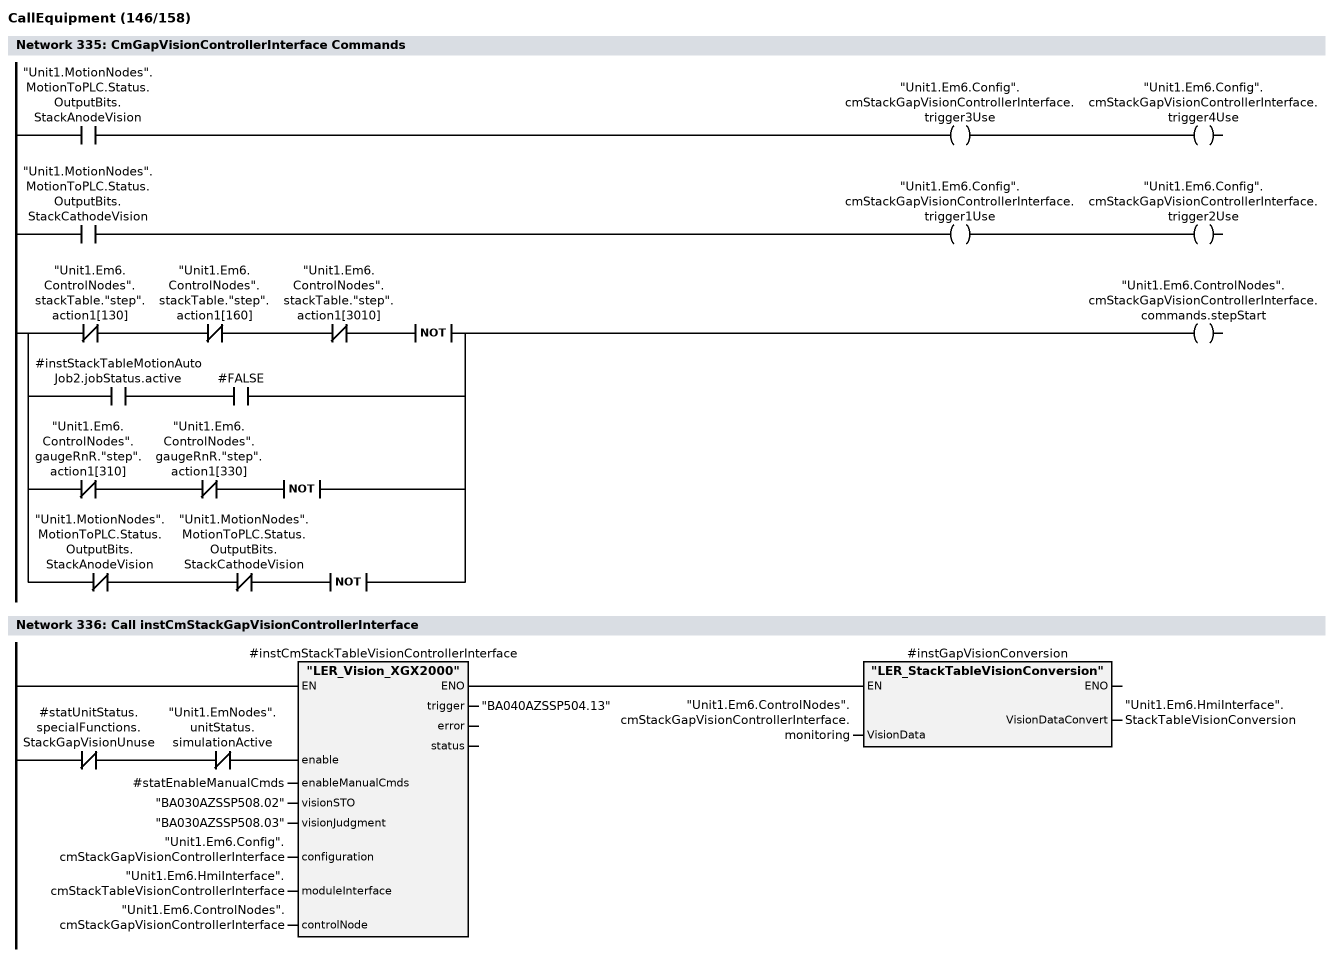
   RUNG wire#powerrail
      Contact( "Unit1.MotionNodes".MotionToPLC.Status.OutputBits.StackAnodeVision )
      Coil( "Unit1.Em6.Config".cmStackGapVisionControllerInterface.trigger3Use )
      Coil( "Unit1.Em6.Config".cmStackGapVisionControllerInterface.trigger4Use )
   END_RUNG
   RUNG wire#powerrail
      Contact( "Unit1.MotionNodes".MotionToPLC.Status.OutputBits.StackCathodeVision )
      Coil( "Unit1.Em6.Config".cmStackGapVisionControllerInterface.trigger1Use )
      Coil( "Unit1.Em6.Config".cmStackGapVisionControllerInterface.trigger2Use )
   END_RUNG
   RUNG wire#powerrail
      I_Contact( "Unit1.Em6.ControlNodes".stackTable."step".action1[130] )
      I_Contact( "Unit1.Em6.ControlNodes".stackTable."step".action1[160] )
      I_Contact( "Unit1.Em6.ControlNodes".stackTable."step".action1[3010] )
      Not()
      wire#w1
      Coil( "Unit1.Em6.ControlNodes".cmStackGapVisionControllerInterface.commands.stepStart )
   END_RUNG
   RUNG wire#powerrail
      Contact( #instStackTableMotionAutoJob2.jobStatus.active )
      Contact( #FALSE )
   END_RUNG wire#w1
   RUNG wire#powerrail
      I_Contact( "Unit1.Em6.ControlNodes".gaugeRnR."step".action1[310] )
      I_Contact( "Unit1.Em6.ControlNodes".gaugeRnR."step".action1[330] )
      Not()
   END_RUNG wire#w1
   RUNG wire#powerrail
      I_Contact( "Unit1.MotionNodes".MotionToPLC.Status.OutputBits.StackAnodeVision )
      I_Contact( "Unit1.MotionNodes".MotionToPLC.Status.OutputBits.StackCathodeVision )
      Not()
   END_RUNG wire#w1
   // the same network as SCL:
   "Unit1.Em6.Config".cmStackGapVisionControllerInterface.trigger3Use := "Unit1.MotionNodes".MotionToPLC.Status.OutputBits.StackAnodeVision;
   "Unit1.Em6.Config".cmStackGapVisionControllerInterface.trigger4Use := "Unit1.MotionNodes".MotionToPLC.Status.OutputBits.StackAnodeVision;
   "Unit1.Em6.Config".cmStackGapVisionControllerInterface.trigger1Use := "Unit1.MotionNodes".MotionToPLC.Status.OutputBits.StackCathodeVision;
   "Unit1.Em6.Config".cmStackGapVisionControllerInterface.trigger2Use := "Unit1.MotionNodes".MotionToPLC.Status.OutputBits.StackCathodeVision;
   "Unit1.Em6.ControlNodes".cmStackGapVisionControllerInterface.commands.stepStart := NOT (NOT "Unit1.Em6.ControlNodes".stackTable."step".action1[130] AND NOT "Unit1.Em6.ControlNodes".stackTable."step".action1[160] AND NOT "Unit1.Em6.ControlNodes".stackTable."step".action1[3010]) OR (#instStackTableMotionAutoJob2.jobStatus.active AND #FALSE) OR NOT (NOT "Unit1.Em6.ControlNodes".gaugeRnR."step".action1[310] AND NOT "Unit1.Em6.ControlNodes".gaugeRnR."step".action1[330]) OR NOT (NOT "Unit1.MotionNodes".MotionToPLC.Status.OutputBits.StackAnodeVision AND NOT "Unit1.MotionNodes".MotionToPLC.Status.OutputBits.StackCathodeVision);
END_REGION

REGION Network 336: Call instCmStackGapVisionControllerInterface
   RUNG wire#powerrail
      #instCmStackTableVisionControllerInterface(enable := wire#w1, enableManualCmds := #statEnableManualCmds, visionSTO := "BA030AZSSP508.02", visionJudgment := "BA030AZSSP508.03", configuration := "Unit1.Em6.Config".cmStackGapVisionControllerInterface, moduleInterface := "Unit1.Em6.HmiInterface".cmStackTableVisionControllerInterface, controlNode := "Unit1.Em6.ControlNodes".cmStackGapVisionControllerInterface, trigger => "BA040AZSSP504.13", error =>, status =>)
      #instGapVisionConversion(VisionData := "Unit1.Em6.ControlNodes".cmStackGapVisionControllerInterface.monitoring, VisionDataConvert => "Unit1.Em6.HmiInterface".StackTableVisionConversion)
   END_RUNG
   RUNG wire#powerrail
      I_Contact( #statUnitStatus.specialFunctions.StackGapVisionUnuse )
      I_Contact( "Unit1.EmNodes".unitStatus.simulationActive )
   END_RUNG wire#w1
   // the same network as SCL:
   #instCmStackTableVisionControllerInterface(enable := NOT #statUnitStatus.specialFunctions.StackGapVisionUnuse AND NOT "Unit1.EmNodes".unitStatus.simulationActive,   // "LER_Vision_XGX2000"
                           enableManualCmds := #statEnableManualCmds,
                           visionSTO := "BA030AZSSP508.02",
                           visionJudgment := "BA030AZSSP508.03",
                           configuration := "Unit1.Em6.Config".cmStackGapVisionControllerInterface,
                           moduleInterface := "Unit1.Em6.HmiInterface".cmStackTableVisionControllerInterface,
                           controlNode := "Unit1.Em6.ControlNodes".cmStackGapVisionControllerInterface,
                           trigger => "BA040AZSSP504.13",
                           ENO => #_w1);
   IF #_w1 THEN
       #instGapVisionConversion(VisionData := "Unit1.Em6.ControlNodes".cmStackGapVisionControllerInterface.monitoring,   // "LER_StackTableVisionConversion"
                               VisionDataConvert => "Unit1.Em6.HmiInterface".StackTableVisionConversion);
   END_IF;
END_REGION

REGION Network 337: *************** Feedback to Unit ***************************
END_REGION

REGION Network 338: Determine StateComplete (SC) in Mode Production
   // Conditions for the Equipment Modules "stateComplete" feedback to the unit. This feedback is given when the task in for the respective state is complete.
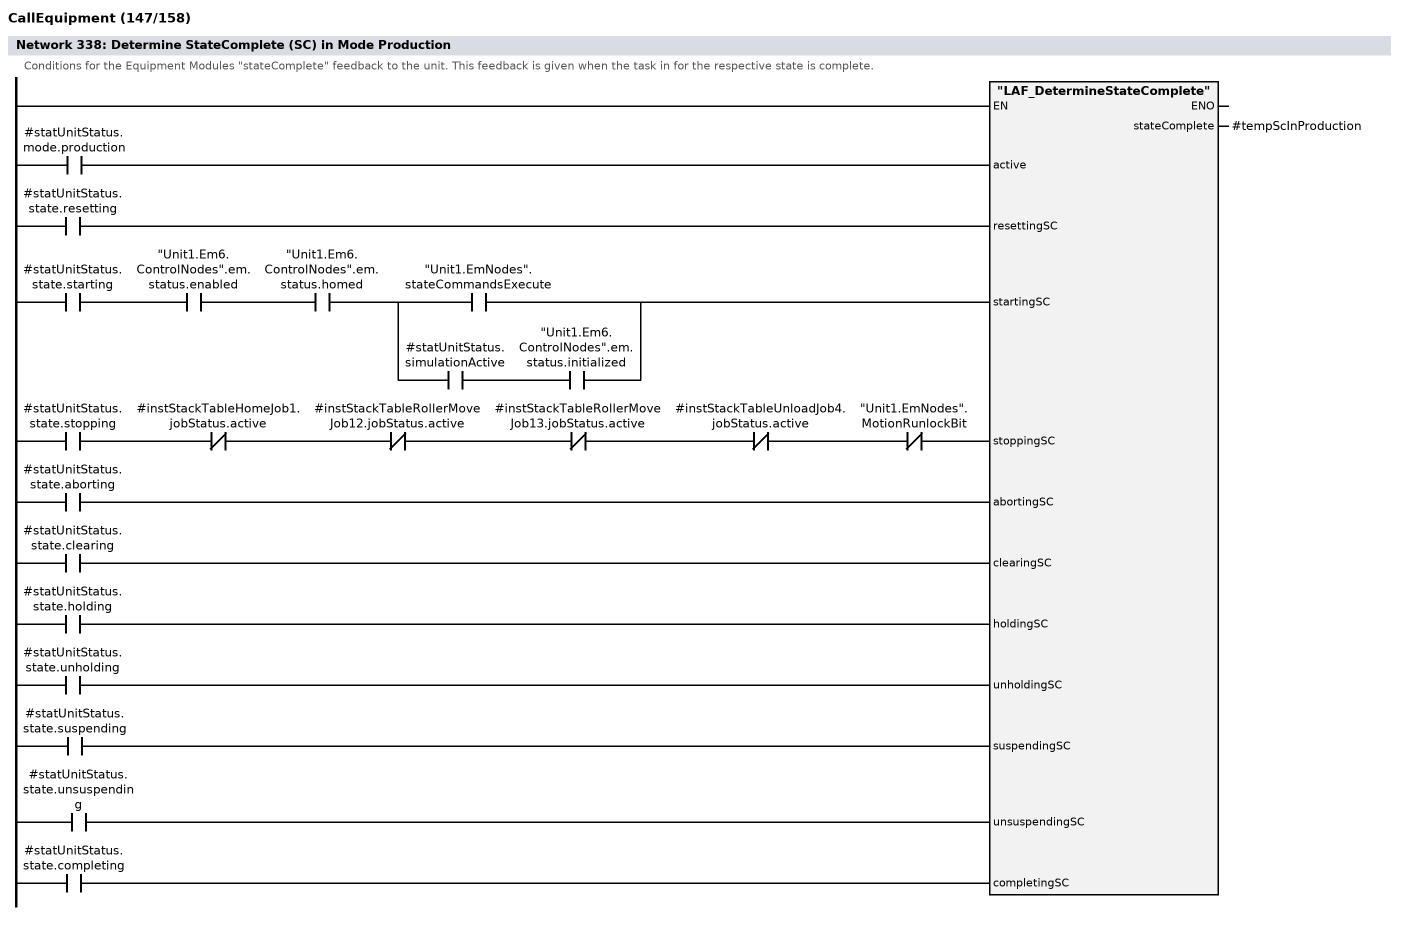
   RUNG wire#powerrail
      "LAF_DetermineStateComplete"(active := wire#w1, resettingSC := wire#w2, startingSC := wire#w4, stoppingSC := wire#w5, abortingSC := wire#w6, clearingSC := wire#w7, holdingSC := wire#w8, unholdingSC := wire#w9, suspendingSC := wire#w10, unsuspendingSC := wire#w11, completingSC := wire#w12, stateComplete => #tempScInProduction)
   END_RUNG
   RUNG wire#powerrail
      Contact( #statUnitStatus.mode.production )
   END_RUNG wire#w1
   RUNG wire#powerrail
      Contact( #statUnitStatus.state.resetting )
   END_RUNG wire#w2
   RUNG wire#powerrail
      Contact( #statUnitStatus.state.starting )
      Contact( "Unit1.Em6.ControlNodes".em.status.enabled )
      Contact( "Unit1.Em6.ControlNodes".em.status.homed )
      wire#w3
      Contact( "Unit1.EmNodes".stateCommandsExecute )
   END_RUNG wire#w4
   RUNG wire#w3
      Contact( #statUnitStatus.simulationActive )
      Contact( "Unit1.Em6.ControlNodes".em.status.initialized )
   END_RUNG wire#w4
   RUNG wire#powerrail
      Contact( #statUnitStatus.state.stopping )
      I_Contact( #instStackTableHomeJob1.jobStatus.active )
      I_Contact( #instStackTableRollerMoveJob12.jobStatus.active )
      I_Contact( #instStackTableRollerMoveJob13.jobStatus.active )
      I_Contact( #instStackTableUnloadJob4.jobStatus.active )
      I_Contact( "Unit1.EmNodes".MotionRunlockBit )
   END_RUNG wire#w5
   RUNG wire#powerrail
      Contact( #statUnitStatus.state.aborting )
   END_RUNG wire#w6
   RUNG wire#powerrail
      Contact( #statUnitStatus.state.clearing )
   END_RUNG wire#w7
   RUNG wire#powerrail
      Contact( #statUnitStatus.state.holding )
   END_RUNG wire#w8
   RUNG wire#powerrail
      Contact( #statUnitStatus.state.unholding )
   END_RUNG wire#w9
   RUNG wire#powerrail
      Contact( #statUnitStatus.state.suspending )
   END_RUNG wire#w10
   RUNG wire#powerrail
      Contact( #statUnitStatus.state.unsuspending )
   END_RUNG wire#w11
   RUNG wire#powerrail
      Contact( #statUnitStatus.state.completing )
   END_RUNG wire#w12
   // the same network as SCL:
   "LAF_DetermineStateComplete"(active := #statUnitStatus.mode.production,
                           resettingSC := #statUnitStatus.state.resetting,
                           startingSC := #statUnitStatus.state.starting AND "Unit1.Em6.ControlNodes".em.status.enabled AND "Unit1.Em6.ControlNodes".em.status.homed AND ("Unit1.EmNodes".stateCommandsExecute OR (#statUnitStatus.simulationActive AND "Unit1.Em6.ControlNodes".em.status.initialized)),
                           stoppingSC := #statUnitStatus.state.stopping AND NOT #instStackTableHomeJob1.jobStatus.active AND NOT #instStackTableRollerMoveJob12.jobStatus.active AND NOT #instStackTableRollerMoveJob13.jobStatus.active AND NOT #instStackTableUnloadJob4.jobStatus.active AND NOT "Unit1.EmNodes".MotionRunlockBit,
                           abortingSC := #statUnitStatus.state.aborting,
                           clearingSC := #statUnitStatus.state.clearing,
                           holdingSC := #statUnitStatus.state.holding,
                           unholdingSC := #statUnitStatus.state.unholding,
                           suspendingSC := #statUnitStatus.state.suspending,
                           unsuspendingSC := #statUnitStatus.state.unsuspending,
                           completingSC := #statUnitStatus.state.completing,
                           stateComplete => #tempScInProduction);
END_REGION

REGION Network 339: Determine StateComplete (SC) in Mode Maintenance/Manual
   // Conditions for the Equipment Modules "stateComplete" feedback to the unit. This feedback is given when the task in for the respective state is complete.
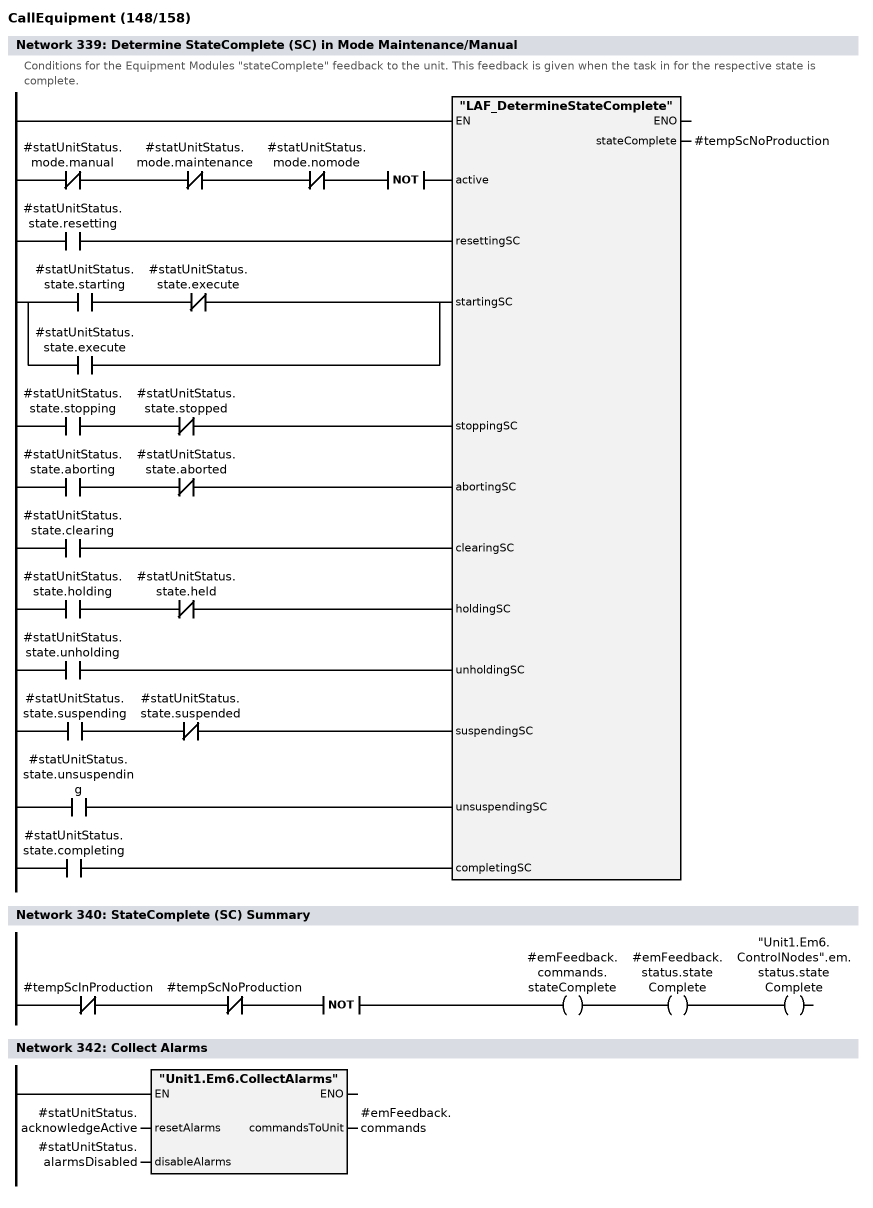
   RUNG wire#powerrail
      "LAF_DetermineStateComplete"(active := wire#w1, resettingSC := wire#w2, startingSC := wire#w3, stoppingSC := wire#w4, abortingSC := wire#w5, clearingSC := wire#w6, holdingSC := wire#w7, unholdingSC := wire#w8, suspendingSC := wire#w9, unsuspendingSC := wire#w10, completingSC := wire#w11, stateComplete => #tempScNoProduction)
   END_RUNG
   RUNG wire#powerrail
      I_Contact( #statUnitStatus.mode.manual )
      I_Contact( #statUnitStatus.mode.maintenance )
      I_Contact( #statUnitStatus.mode.nomode )
      Not()
   END_RUNG wire#w1
   RUNG wire#powerrail
      Contact( #statUnitStatus.state.resetting )
   END_RUNG wire#w2
   RUNG wire#powerrail
      Contact( #statUnitStatus.state.starting )
      I_Contact( #statUnitStatus.state.execute )
   END_RUNG wire#w3
   RUNG wire#powerrail
      Contact( #statUnitStatus.state.execute )
   END_RUNG wire#w3
   RUNG wire#powerrail
      Contact( #statUnitStatus.state.stopping )
      I_Contact( #statUnitStatus.state.stopped )
   END_RUNG wire#w4
   RUNG wire#powerrail
      Contact( #statUnitStatus.state.aborting )
      I_Contact( #statUnitStatus.state.aborted )
   END_RUNG wire#w5
   RUNG wire#powerrail
      Contact( #statUnitStatus.state.clearing )
   END_RUNG wire#w6
   RUNG wire#powerrail
      Contact( #statUnitStatus.state.holding )
      I_Contact( #statUnitStatus.state.held )
   END_RUNG wire#w7
   RUNG wire#powerrail
      Contact( #statUnitStatus.state.unholding )
   END_RUNG wire#w8
   RUNG wire#powerrail
      Contact( #statUnitStatus.state.suspending )
      I_Contact( #statUnitStatus.state.suspended )
   END_RUNG wire#w9
   RUNG wire#powerrail
      Contact( #statUnitStatus.state.unsuspending )
   END_RUNG wire#w10
   RUNG wire#powerrail
      Contact( #statUnitStatus.state.completing )
   END_RUNG wire#w11
   // the same network as SCL:
   "LAF_DetermineStateComplete"(active := NOT (NOT #statUnitStatus.mode.manual AND NOT #statUnitStatus.mode.maintenance AND NOT #statUnitStatus.mode.nomode),
                           resettingSC := #statUnitStatus.state.resetting,
                           startingSC := (#statUnitStatus.state.starting AND NOT #statUnitStatus.state.execute) OR #statUnitStatus.state.execute,
                           stoppingSC := #statUnitStatus.state.stopping AND NOT #statUnitStatus.state.stopped,
                           abortingSC := #statUnitStatus.state.aborting AND NOT #statUnitStatus.state.aborted,
                           clearingSC := #statUnitStatus.state.clearing,
                           holdingSC := #statUnitStatus.state.holding AND NOT #statUnitStatus.state.held,
                           unholdingSC := #statUnitStatus.state.unholding,
                           suspendingSC := #statUnitStatus.state.suspending AND NOT #statUnitStatus.state.suspended,
                           unsuspendingSC := #statUnitStatus.state.unsuspending,
                           completingSC := #statUnitStatus.state.completing,
                           stateComplete => #tempScNoProduction);
END_REGION

REGION Network 340: StateComplete (SC) Summary
   RUNG wire#powerrail
      I_Contact( #tempScInProduction )
      I_Contact( #tempScNoProduction )
      Not()
      Coil( #emFeedback.commands.stateComplete )
      Coil( #emFeedback.status.stateComplete )
      Coil( "Unit1.Em6.ControlNodes".em.status.stateComplete )
   END_RUNG
   // the same network as SCL:
   #emFeedback.commands.stateComplete := NOT (NOT #tempScInProduction AND NOT #tempScNoProduction);
   #emFeedback.status.stateComplete := #emFeedback.commands.stateComplete;
   "Unit1.Em6.ControlNodes".em.status.stateComplete := #emFeedback.commands.stateComplete;
END_REGION

REGION Network 341: *************** Alarms **********************************
END_REGION

REGION Network 342: Collect Alarms
   RUNG wire#powerrail
      "Unit1.Em6.CollectAlarms"(resetAlarms := #statUnitStatus.acknowledgeActive, disableAlarms := #statUnitStatus.alarmsDisabled, commandsToUnit => #emFeedback.commands)
   END_RUNG
   // the same network as SCL:
   "Unit1.Em6.CollectAlarms"(resetAlarms := #statUnitStatus.acknowledgeActive,
                           disableAlarms := #statUnitStatus.alarmsDisabled,
                           commandsToUnit => #emFeedback.commands);
END_REGION

REGION Network 343: Manage Alarms
   // Derive commands from the ProDiag supervision. The ProDiag supervisions contain categories which define the reaction of these supervisions (e.g. abort, stop, hold). These are handed over as commands to the unit level.
   // Alternatively, if no ProDiag should be used, you can use the LAF_ManageBitAlarms to realize bit alarm handling. This block can be found in LAF in folder 70_AlarmHandling.
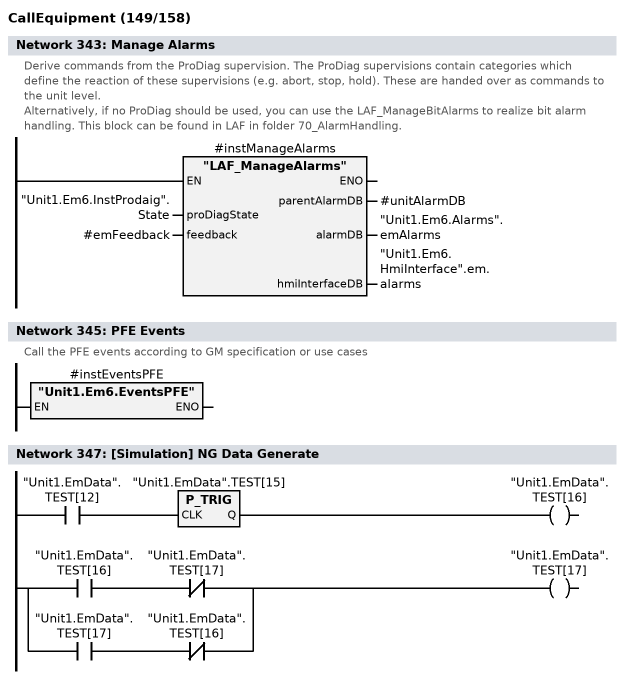
   RUNG wire#powerrail
      #instManageAlarms(proDiagState := "Unit1.Em6.InstProdaig".State, feedback := #emFeedback, parentAlarmDB => #unitAlarmDB, alarmDB => "Unit1.Em6.Alarms".emAlarms, hmiInterfaceDB => "Unit1.Em6.HmiInterface".em.alarms)
   END_RUNG
   // the same network as SCL:
   #instManageAlarms(proDiagState := "Unit1.Em6.InstProdaig".State,   // "LAF_ManageAlarms"
                     feedback := #emFeedback,
                     parentAlarmDB => #unitAlarmDB,
                     alarmDB => "Unit1.Em6.Alarms".emAlarms,
                     hmiInterfaceDB => "Unit1.Em6.HmiInterface".em.alarms);
END_REGION

REGION Network 344: *************** PFE Events**********************************
END_REGION

REGION Network 345: PFE Events
   // Call the PFE events according to GM specification or use cases
   RUNG wire#powerrail
      #instEventsPFE()
   END_RUNG
   // the same network as SCL:
   #instEventsPFE();   // "Unit1.Em6.EventsPFE"
END_REGION

REGION Network 346: ******************** Part Data ********************
END_REGION

REGION Network 347: [Simulation] NG Data Generate
   RUNG wire#powerrail
      Contact( "Unit1.EmData".TEST[12] )
      P_Trig( "Unit1.EmData".TEST[15] )
      Coil( "Unit1.EmData".TEST[16] )
   END_RUNG
   RUNG wire#powerrail
      Contact( "Unit1.EmData".TEST[16] )
      I_Contact( "Unit1.EmData".TEST[17] )
      wire#w1
      Coil( "Unit1.EmData".TEST[17] )
   END_RUNG
   RUNG wire#powerrail
      Contact( "Unit1.EmData".TEST[17] )
      I_Contact( "Unit1.EmData".TEST[16] )
   END_RUNG wire#w1
   // the same network as SCL:
   #_w1 := "Unit1.EmData".TEST[12];
   #_w2 := #_w1 AND NOT "Unit1.EmData".TEST[15];   // rising edge
   "Unit1.EmData".TEST[15] := #_w1;
   "Unit1.EmData".TEST[16] := #_w2;
   "Unit1.EmData".TEST[17] := ("Unit1.EmData".TEST[16] AND NOT "Unit1.EmData".TEST[17]) OR ("Unit1.EmData".TEST[17] AND NOT "Unit1.EmData".TEST[16]);
END_REGION

REGION Network 348: Gap Vision Data
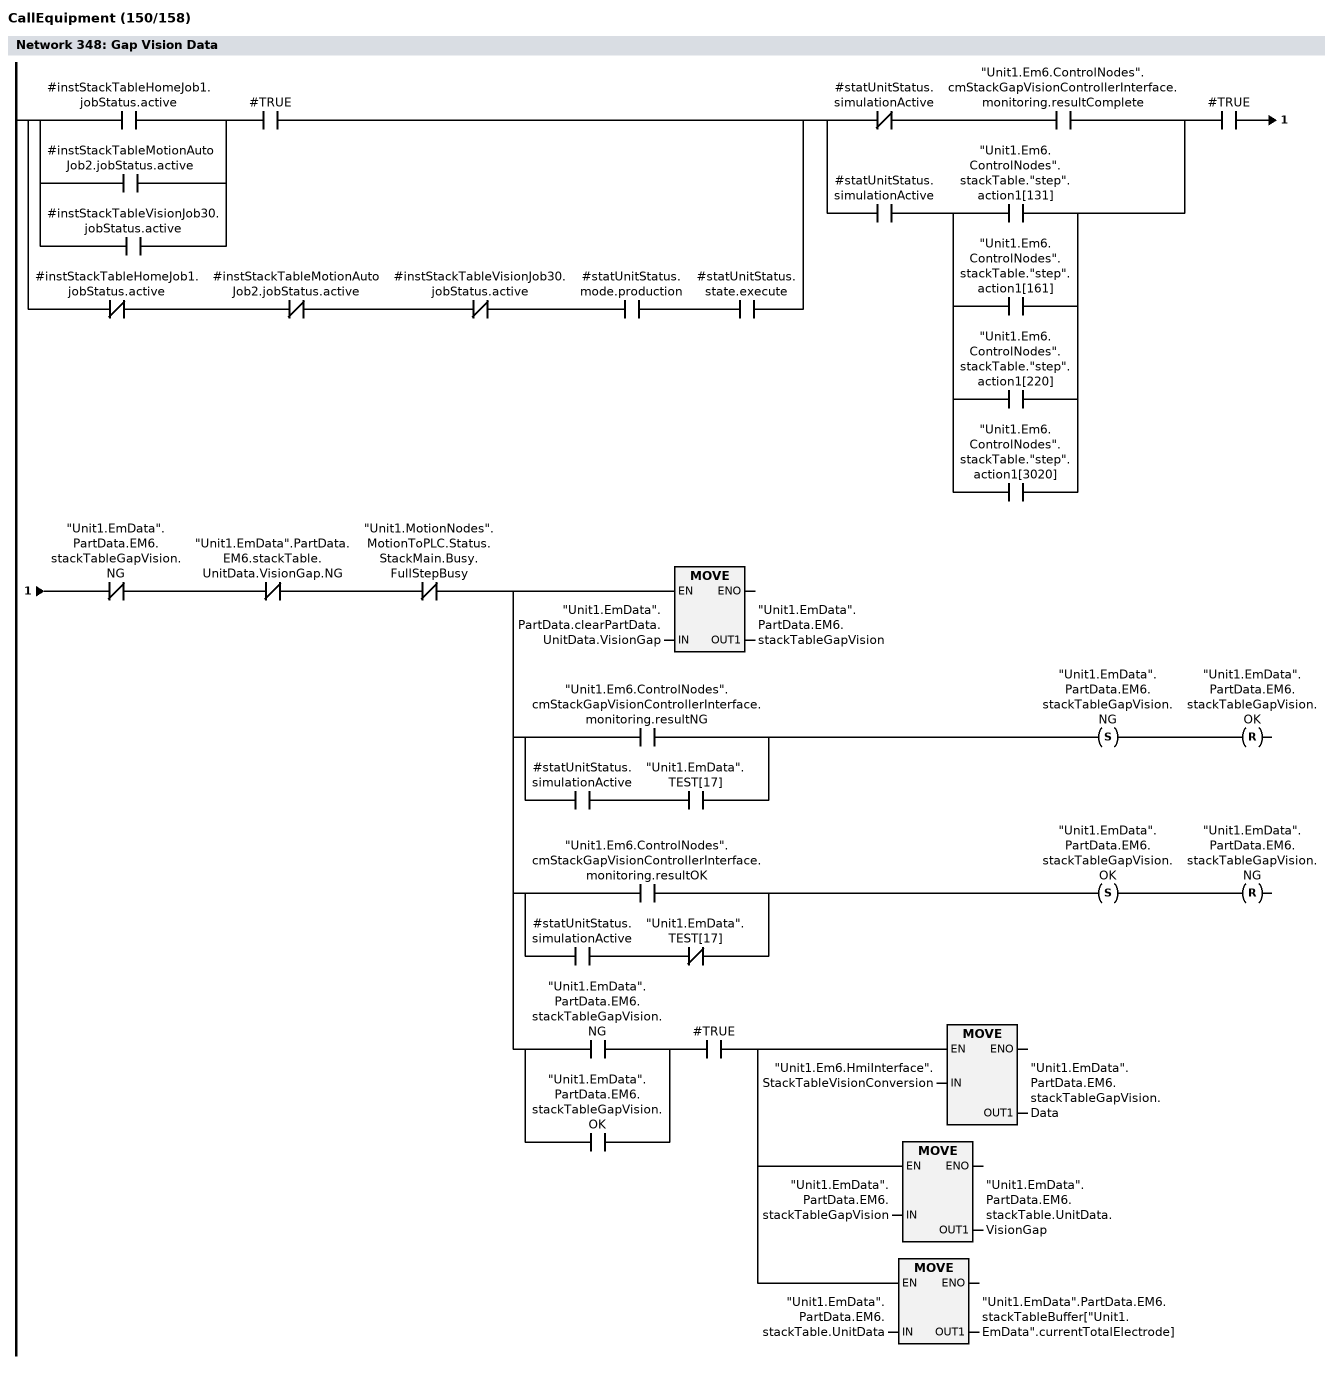
   RUNG wire#powerrail
      Contact( #instStackTableHomeJob1.jobStatus.active )
      wire#w1
      Contact( #TRUE )
      wire#w2
      I_Contact( #statUnitStatus.simulationActive )
      Contact( "Unit1.Em6.ControlNodes".cmStackGapVisionControllerInterface.monitoring.resultComplete )
      wire#w3
      Contact( #TRUE )
      I_Contact( "Unit1.EmData".PartData.EM6.stackTableGapVision.NG )
      I_Contact( "Unit1.EmData".PartData.EM6.stackTable.UnitData.VisionGap.NG )
      I_Contact( "Unit1.MotionNodes".MotionToPLC.Status.StackMain.Busy.FullStepBusy )
      wire#w5
      Move(in := "Unit1.EmData".PartData.clearPartData.UnitData.VisionGap, out1 => "Unit1.EmData".PartData.EM6.stackTableGapVision)
   END_RUNG
   RUNG wire#powerrail
      Contact( #instStackTableMotionAutoJob2.jobStatus.active )
   END_RUNG wire#w1
   RUNG wire#powerrail
      Contact( #instStackTableVisionJob30.jobStatus.active )
   END_RUNG wire#w1
   RUNG wire#powerrail
      I_Contact( #instStackTableHomeJob1.jobStatus.active )
      I_Contact( #instStackTableMotionAutoJob2.jobStatus.active )
      I_Contact( #instStackTableVisionJob30.jobStatus.active )
      Contact( #statUnitStatus.mode.production )
      Contact( #statUnitStatus.state.execute )
   END_RUNG wire#w2
   RUNG wire#w2
      Contact( #statUnitStatus.simulationActive )
      wire#w4
      Contact( "Unit1.Em6.ControlNodes".stackTable."step".action1[131] )
   END_RUNG wire#w3
   RUNG wire#w4
      Contact( "Unit1.Em6.ControlNodes".stackTable."step".action1[161] )
   END_RUNG wire#w3
   RUNG wire#w4
      Contact( "Unit1.Em6.ControlNodes".stackTable."step".action1[220] )
   END_RUNG wire#w3
   RUNG wire#w4
      Contact( "Unit1.Em6.ControlNodes".stackTable."step".action1[3020] )
   END_RUNG wire#w3
   RUNG wire#w5
      Contact( "Unit1.Em6.ControlNodes".cmStackGapVisionControllerInterface.monitoring.resultNG )
      wire#w6
      S_Coil( "Unit1.EmData".PartData.EM6.stackTableGapVision.NG )
      R_Coil( "Unit1.EmData".PartData.EM6.stackTableGapVision.OK )
   END_RUNG
   RUNG wire#w5
      Contact( #statUnitStatus.simulationActive )
      Contact( "Unit1.EmData".TEST[17] )
   END_RUNG wire#w6
   RUNG wire#w5
      Contact( "Unit1.Em6.ControlNodes".cmStackGapVisionControllerInterface.monitoring.resultOK )
      wire#w7
      S_Coil( "Unit1.EmData".PartData.EM6.stackTableGapVision.OK )
      R_Coil( "Unit1.EmData".PartData.EM6.stackTableGapVision.NG )
   END_RUNG
   RUNG wire#w5
      Contact( #statUnitStatus.simulationActive )
      I_Contact( "Unit1.EmData".TEST[17] )
   END_RUNG wire#w7
   RUNG wire#w5
      Contact( "Unit1.EmData".PartData.EM6.stackTableGapVision.NG )
      wire#w8
      Contact( #TRUE )
      wire#w9
      Move(in := "Unit1.Em6.HmiInterface".StackTableVisionConversion, out1 => "Unit1.EmData".PartData.EM6.stackTableGapVision.Data)
   END_RUNG
   RUNG wire#w5
      Contact( "Unit1.EmData".PartData.EM6.stackTableGapVision.OK )
   END_RUNG wire#w8
   RUNG wire#w9
      Move(in := "Unit1.EmData".PartData.EM6.stackTableGapVision, out1 => "Unit1.EmData".PartData.EM6.stackTable.UnitData.VisionGap)
   END_RUNG
   RUNG wire#w9
      Move(in := "Unit1.EmData".PartData.EM6.stackTable.UnitData, out1 => "Unit1.EmData".PartData.EM6.stackTableBuffer["Unit1.EmData".currentTotalElectrode])
   END_RUNG
   // the same network as SCL:
   #_w1 := (((#instStackTableHomeJob1.jobStatus.active OR #instStackTableMotionAutoJob2.jobStatus.active OR #instStackTableVisionJob30.jobStatus.active) AND #TRUE) OR (NOT #instStackTableHomeJob1.jobStatus.active AND NOT #instStackTableMotionAutoJob2.jobStatus.active AND NOT #instStackTableVisionJob30.jobStatus.active AND #statUnitStatus.mode.production AND #statUnitStatus.state.execute)) AND ((NOT #statUnitStatus.simulationActive AND "Unit1.Em6.ControlNodes".cmStackGapVisionControllerInterface.monitoring.resultComplete) OR (#statUnitStatus.simulationActive AND ("Unit1.Em6.ControlNodes".stackTable."step".action1[131] OR "Unit1.Em6.ControlNodes".stackTable."step".action1[161] OR "Unit1.Em6.ControlNodes".stackTable."step".action1[220] OR "Unit1.Em6.ControlNodes".stackTable."step".action1[3020]))) AND #TRUE AND NOT "Unit1.EmData".PartData.EM6.stackTableGapVision.NG AND NOT "Unit1.EmData".PartData.EM6.stackTable.UnitData.VisionGap.NG AND NOT "Unit1.MotionNodes".MotionToPLC.Status.StackMain.Busy.FullStepBusy;
   IF #_w1 THEN
       "Unit1.EmData".PartData.EM6.stackTableGapVision := "Unit1.EmData".PartData.clearPartData.UnitData.VisionGap;
   END_IF;
   IF #_w1 AND ("Unit1.Em6.ControlNodes".cmStackGapVisionControllerInterface.monitoring.resultNG OR (#statUnitStatus.simulationActive AND "Unit1.EmData".TEST[17])) THEN
       "Unit1.EmData".PartData.EM6.stackTableGapVision.NG := TRUE;
       "Unit1.EmData".PartData.EM6.stackTableGapVision.OK := FALSE;
   END_IF;
   IF #_w1 AND ("Unit1.Em6.ControlNodes".cmStackGapVisionControllerInterface.monitoring.resultOK OR (#statUnitStatus.simulationActive AND NOT "Unit1.EmData".TEST[17])) THEN
       "Unit1.EmData".PartData.EM6.stackTableGapVision.OK := TRUE;
       "Unit1.EmData".PartData.EM6.stackTableGapVision.NG := FALSE;
   END_IF;
   IF #_w1 AND ("Unit1.EmData".PartData.EM6.stackTableGapVision.NG OR "Unit1.EmData".PartData.EM6.stackTableGapVision.OK) AND #TRUE THEN
       "Unit1.EmData".PartData.EM6.stackTableGapVision.Data := "Unit1.Em6.HmiInterface".StackTableVisionConversion;
       "Unit1.EmData".PartData.EM6.stackTable.UnitData.VisionGap := "Unit1.EmData".PartData.EM6.stackTableGapVision;
       "Unit1.EmData".PartData.EM6.stackTableBuffer["Unit1.EmData".currentTotalElectrode] := "Unit1.EmData".PartData.EM6.stackTable.UnitData;
   END_IF;
END_REGION

REGION Network 349: ******************** Map 64Pos Positiotion ********************
END_REGION

REGION Network 350: StackTableAxis Z Postion [1] Mapping
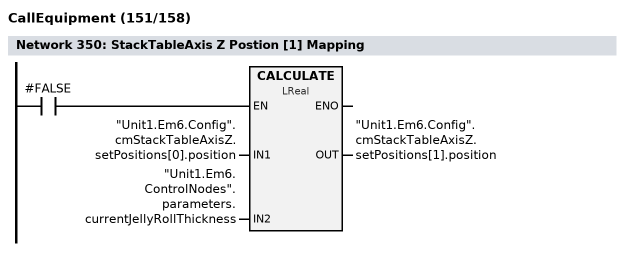
   RUNG wire#powerrail
      Contact( #FALSE )
      { S7_Templates := "SrcType := LReal"; S7_Expression := "IN1 + IN2" } Calculate(in1 := "Unit1.Em6.Config".cmStackTableAxisZ.setPositions[0].position, in2 := "Unit1.Em6.ControlNodes".parameters.currentJellyRollThickness, out => "Unit1.Em6.Config".cmStackTableAxisZ.setPositions[1].position)
   END_RUNG
   // the same network as SCL:
   IF #FALSE THEN
       "Unit1.Em6.Config".cmStackTableAxisZ.setPositions[1].position := "Unit1.Em6.Config".cmStackTableAxisZ.setPositions[0].position + "Unit1.Em6.ControlNodes".parameters.currentJellyRollThickness;
   END_IF;
END_REGION

REGION Network 351: ******************** Unit Output ********************
END_REGION

REGION Network 352: Em Nodes Brake Test
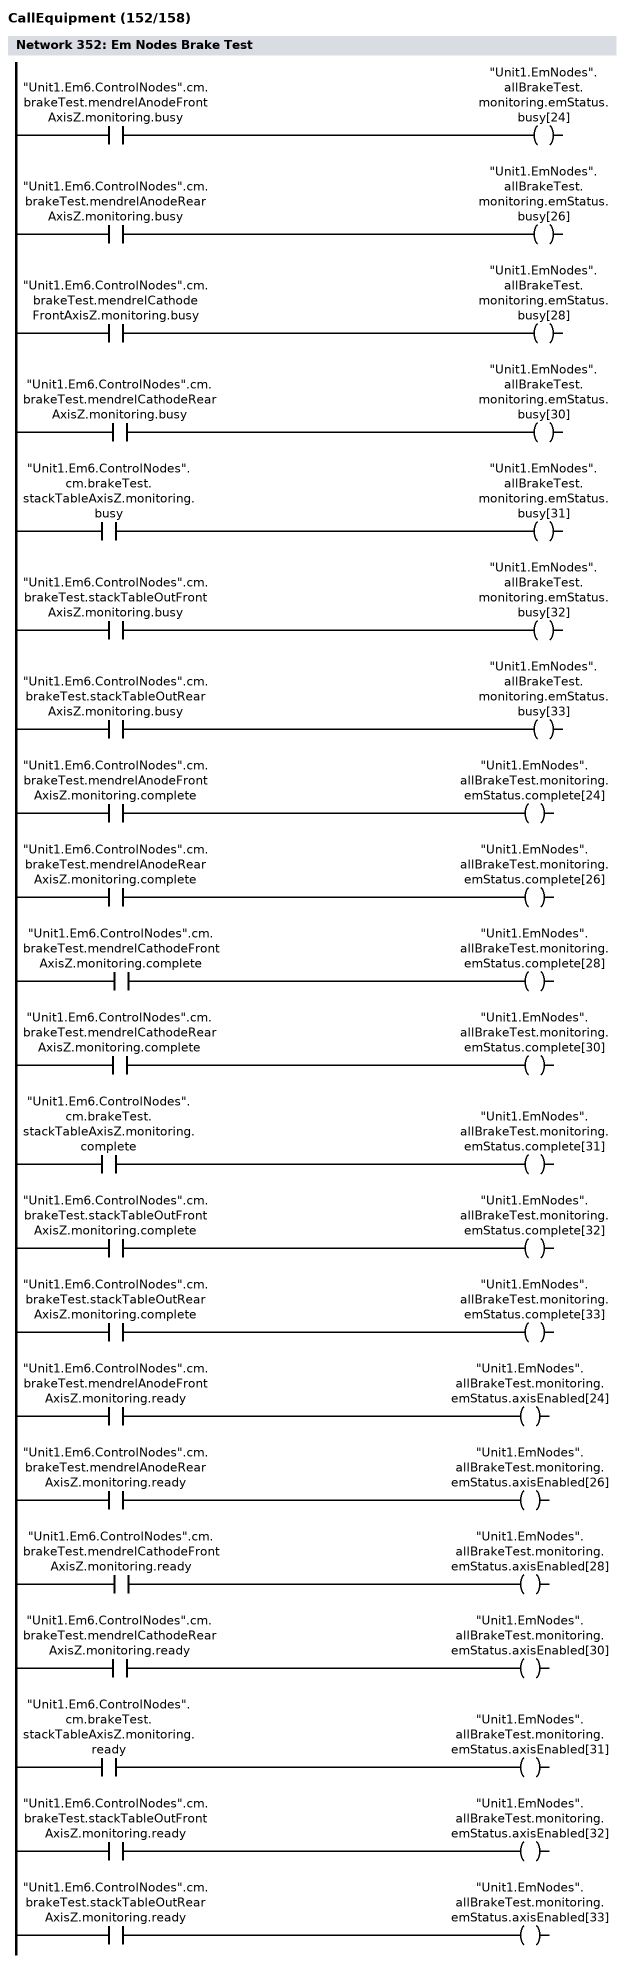
   RUNG wire#powerrail
      Contact( "Unit1.Em6.ControlNodes".cm.brakeTest.mendrelAnodeFrontAxisZ.monitoring.busy )
      Coil( "Unit1.EmNodes".allBrakeTest.monitoring.emStatus.busy[24] )
   END_RUNG
   RUNG wire#powerrail
      Contact( "Unit1.Em6.ControlNodes".cm.brakeTest.mendrelAnodeRearAxisZ.monitoring.busy )
      Coil( "Unit1.EmNodes".allBrakeTest.monitoring.emStatus.busy[26] )
   END_RUNG
   RUNG wire#powerrail
      Contact( "Unit1.Em6.ControlNodes".cm.brakeTest.mendrelCathodeFrontAxisZ.monitoring.busy )
      Coil( "Unit1.EmNodes".allBrakeTest.monitoring.emStatus.busy[28] )
   END_RUNG
   RUNG wire#powerrail
      Contact( "Unit1.Em6.ControlNodes".cm.brakeTest.mendrelCathodeRearAxisZ.monitoring.busy )
      Coil( "Unit1.EmNodes".allBrakeTest.monitoring.emStatus.busy[30] )
   END_RUNG
   RUNG wire#powerrail
      Contact( "Unit1.Em6.ControlNodes".cm.brakeTest.stackTableAxisZ.monitoring.busy )
      Coil( "Unit1.EmNodes".allBrakeTest.monitoring.emStatus.busy[31] )
   END_RUNG
   RUNG wire#powerrail
      Contact( "Unit1.Em6.ControlNodes".cm.brakeTest.stackTableOutFrontAxisZ.monitoring.busy )
      Coil( "Unit1.EmNodes".allBrakeTest.monitoring.emStatus.busy[32] )
   END_RUNG
   RUNG wire#powerrail
      Contact( "Unit1.Em6.ControlNodes".cm.brakeTest.stackTableOutRearAxisZ.monitoring.busy )
      Coil( "Unit1.EmNodes".allBrakeTest.monitoring.emStatus.busy[33] )
   END_RUNG
   RUNG wire#powerrail
      Contact( "Unit1.Em6.ControlNodes".cm.brakeTest.mendrelAnodeFrontAxisZ.monitoring.complete )
      Coil( "Unit1.EmNodes".allBrakeTest.monitoring.emStatus.complete[24] )
   END_RUNG
   RUNG wire#powerrail
      Contact( "Unit1.Em6.ControlNodes".cm.brakeTest.mendrelAnodeRearAxisZ.monitoring.complete )
      Coil( "Unit1.EmNodes".allBrakeTest.monitoring.emStatus.complete[26] )
   END_RUNG
   RUNG wire#powerrail
      Contact( "Unit1.Em6.ControlNodes".cm.brakeTest.mendrelCathodeFrontAxisZ.monitoring.complete )
      Coil( "Unit1.EmNodes".allBrakeTest.monitoring.emStatus.complete[28] )
   END_RUNG
   RUNG wire#powerrail
      Contact( "Unit1.Em6.ControlNodes".cm.brakeTest.mendrelCathodeRearAxisZ.monitoring.complete )
      Coil( "Unit1.EmNodes".allBrakeTest.monitoring.emStatus.complete[30] )
   END_RUNG
   RUNG wire#powerrail
      Contact( "Unit1.Em6.ControlNodes".cm.brakeTest.stackTableAxisZ.monitoring.complete )
      Coil( "Unit1.EmNodes".allBrakeTest.monitoring.emStatus.complete[31] )
   END_RUNG
   RUNG wire#powerrail
      Contact( "Unit1.Em6.ControlNodes".cm.brakeTest.stackTableOutFrontAxisZ.monitoring.complete )
      Coil( "Unit1.EmNodes".allBrakeTest.monitoring.emStatus.complete[32] )
   END_RUNG
   RUNG wire#powerrail
      Contact( "Unit1.Em6.ControlNodes".cm.brakeTest.stackTableOutRearAxisZ.monitoring.complete )
      Coil( "Unit1.EmNodes".allBrakeTest.monitoring.emStatus.complete[33] )
   END_RUNG
   RUNG wire#powerrail
      Contact( "Unit1.Em6.ControlNodes".cm.brakeTest.mendrelAnodeFrontAxisZ.monitoring.ready )
      Coil( "Unit1.EmNodes".allBrakeTest.monitoring.emStatus.axisEnabled[24] )
   END_RUNG
   RUNG wire#powerrail
      Contact( "Unit1.Em6.ControlNodes".cm.brakeTest.mendrelAnodeRearAxisZ.monitoring.ready )
      Coil( "Unit1.EmNodes".allBrakeTest.monitoring.emStatus.axisEnabled[26] )
   END_RUNG
   RUNG wire#powerrail
      Contact( "Unit1.Em6.ControlNodes".cm.brakeTest.mendrelCathodeFrontAxisZ.monitoring.ready )
      Coil( "Unit1.EmNodes".allBrakeTest.monitoring.emStatus.axisEnabled[28] )
   END_RUNG
   RUNG wire#powerrail
      Contact( "Unit1.Em6.ControlNodes".cm.brakeTest.mendrelCathodeRearAxisZ.monitoring.ready )
      Coil( "Unit1.EmNodes".allBrakeTest.monitoring.emStatus.axisEnabled[30] )
   END_RUNG
   RUNG wire#powerrail
      Contact( "Unit1.Em6.ControlNodes".cm.brakeTest.stackTableAxisZ.monitoring.ready )
      Coil( "Unit1.EmNodes".allBrakeTest.monitoring.emStatus.axisEnabled[31] )
   END_RUNG
   RUNG wire#powerrail
      Contact( "Unit1.Em6.ControlNodes".cm.brakeTest.stackTableOutFrontAxisZ.monitoring.ready )
      Coil( "Unit1.EmNodes".allBrakeTest.monitoring.emStatus.axisEnabled[32] )
   END_RUNG
   RUNG wire#powerrail
      Contact( "Unit1.Em6.ControlNodes".cm.brakeTest.stackTableOutRearAxisZ.monitoring.ready )
      Coil( "Unit1.EmNodes".allBrakeTest.monitoring.emStatus.axisEnabled[33] )
   END_RUNG
   // the same network as SCL:
   "Unit1.EmNodes".allBrakeTest.monitoring.emStatus.busy[24] := "Unit1.Em6.ControlNodes".cm.brakeTest.mendrelAnodeFrontAxisZ.monitoring.busy;
   "Unit1.EmNodes".allBrakeTest.monitoring.emStatus.busy[26] := "Unit1.Em6.ControlNodes".cm.brakeTest.mendrelAnodeRearAxisZ.monitoring.busy;
   "Unit1.EmNodes".allBrakeTest.monitoring.emStatus.busy[28] := "Unit1.Em6.ControlNodes".cm.brakeTest.mendrelCathodeFrontAxisZ.monitoring.busy;
   "Unit1.EmNodes".allBrakeTest.monitoring.emStatus.busy[30] := "Unit1.Em6.ControlNodes".cm.brakeTest.mendrelCathodeRearAxisZ.monitoring.busy;
   "Unit1.EmNodes".allBrakeTest.monitoring.emStatus.busy[31] := "Unit1.Em6.ControlNodes".cm.brakeTest.stackTableAxisZ.monitoring.busy;
   "Unit1.EmNodes".allBrakeTest.monitoring.emStatus.busy[32] := "Unit1.Em6.ControlNodes".cm.brakeTest.stackTableOutFrontAxisZ.monitoring.busy;
   "Unit1.EmNodes".allBrakeTest.monitoring.emStatus.busy[33] := "Unit1.Em6.ControlNodes".cm.brakeTest.stackTableOutRearAxisZ.monitoring.busy;
   "Unit1.EmNodes".allBrakeTest.monitoring.emStatus.complete[24] := "Unit1.Em6.ControlNodes".cm.brakeTest.mendrelAnodeFrontAxisZ.monitoring.complete;
   "Unit1.EmNodes".allBrakeTest.monitoring.emStatus.complete[26] := "Unit1.Em6.ControlNodes".cm.brakeTest.mendrelAnodeRearAxisZ.monitoring.complete;
   "Unit1.EmNodes".allBrakeTest.monitoring.emStatus.complete[28] := "Unit1.Em6.ControlNodes".cm.brakeTest.mendrelCathodeFrontAxisZ.monitoring.complete;
   "Unit1.EmNodes".allBrakeTest.monitoring.emStatus.complete[30] := "Unit1.Em6.ControlNodes".cm.brakeTest.mendrelCathodeRearAxisZ.monitoring.complete;
   "Unit1.EmNodes".allBrakeTest.monitoring.emStatus.complete[31] := "Unit1.Em6.ControlNodes".cm.brakeTest.stackTableAxisZ.monitoring.complete;
   "Unit1.EmNodes".allBrakeTest.monitoring.emStatus.complete[32] := "Unit1.Em6.ControlNodes".cm.brakeTest.stackTableOutFrontAxisZ.monitoring.complete;
   "Unit1.EmNodes".allBrakeTest.monitoring.emStatus.complete[33] := "Unit1.Em6.ControlNodes".cm.brakeTest.stackTableOutRearAxisZ.monitoring.complete;
   "Unit1.EmNodes".allBrakeTest.monitoring.emStatus.axisEnabled[24] := "Unit1.Em6.ControlNodes".cm.brakeTest.mendrelAnodeFrontAxisZ.monitoring.ready;
   "Unit1.EmNodes".allBrakeTest.monitoring.emStatus.axisEnabled[26] := "Unit1.Em6.ControlNodes".cm.brakeTest.mendrelAnodeRearAxisZ.monitoring.ready;
   "Unit1.EmNodes".allBrakeTest.monitoring.emStatus.axisEnabled[28] := "Unit1.Em6.ControlNodes".cm.brakeTest.mendrelCathodeFrontAxisZ.monitoring.ready;
   "Unit1.EmNodes".allBrakeTest.monitoring.emStatus.axisEnabled[30] := "Unit1.Em6.ControlNodes".cm.brakeTest.mendrelCathodeRearAxisZ.monitoring.ready;
   "Unit1.EmNodes".allBrakeTest.monitoring.emStatus.axisEnabled[31] := "Unit1.Em6.ControlNodes".cm.brakeTest.stackTableAxisZ.monitoring.ready;
   "Unit1.EmNodes".allBrakeTest.monitoring.emStatus.axisEnabled[32] := "Unit1.Em6.ControlNodes".cm.brakeTest.stackTableOutFrontAxisZ.monitoring.ready;
   "Unit1.EmNodes".allBrakeTest.monitoring.emStatus.axisEnabled[33] := "Unit1.Em6.ControlNodes".cm.brakeTest.stackTableOutRearAxisZ.monitoring.ready;
END_REGION

REGION Network 353: Em Relations Home Check
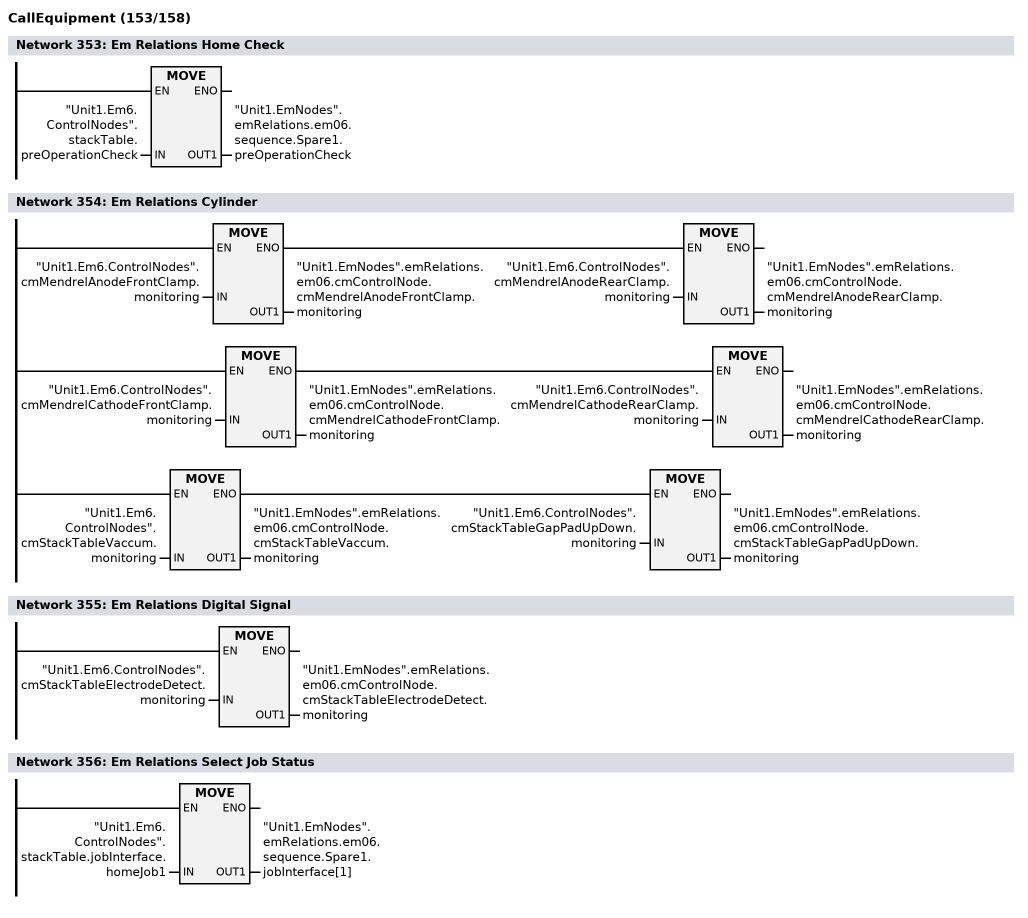
   RUNG wire#powerrail
      Move(in := "Unit1.Em6.ControlNodes".stackTable.preOperationCheck, out1 => "Unit1.EmNodes".emRelations.em06.sequence.Spare1.preOperationCheck)
   END_RUNG
   // the same network as SCL:
   "Unit1.EmNodes".emRelations.em06.sequence.Spare1.preOperationCheck := "Unit1.Em6.ControlNodes".stackTable.preOperationCheck;
END_REGION

REGION Network 354: Em Relations Cylinder
   RUNG wire#powerrail
      Move(in := "Unit1.Em6.ControlNodes".cmMendrelAnodeFrontClamp.monitoring, out1 => "Unit1.EmNodes".emRelations.em06.cmControlNode.cmMendrelAnodeFrontClamp.monitoring)
      Move(in := "Unit1.Em6.ControlNodes".cmMendrelAnodeRearClamp.monitoring, out1 => "Unit1.EmNodes".emRelations.em06.cmControlNode.cmMendrelAnodeRearClamp.monitoring)
   END_RUNG
   RUNG wire#powerrail
      Move(in := "Unit1.Em6.ControlNodes".cmMendrelCathodeFrontClamp.monitoring, out1 => "Unit1.EmNodes".emRelations.em06.cmControlNode.cmMendrelCathodeFrontClamp.monitoring)
      Move(in := "Unit1.Em6.ControlNodes".cmMendrelCathodeRearClamp.monitoring, out1 => "Unit1.EmNodes".emRelations.em06.cmControlNode.cmMendrelCathodeRearClamp.monitoring)
   END_RUNG
   RUNG wire#powerrail
      Move(in := "Unit1.Em6.ControlNodes".cmStackTableVaccum.monitoring, out1 => "Unit1.EmNodes".emRelations.em06.cmControlNode.cmStackTableVaccum.monitoring)
      Move(in := "Unit1.Em6.ControlNodes".cmStackTableGapPadUpDown.monitoring, out1 => "Unit1.EmNodes".emRelations.em06.cmControlNode.cmStackTableGapPadUpDown.monitoring)
   END_RUNG
   // the same network as SCL:
   "Unit1.EmNodes".emRelations.em06.cmControlNode.cmMendrelAnodeFrontClamp.monitoring := "Unit1.Em6.ControlNodes".cmMendrelAnodeFrontClamp.monitoring;
   "Unit1.EmNodes".emRelations.em06.cmControlNode.cmMendrelAnodeRearClamp.monitoring := "Unit1.Em6.ControlNodes".cmMendrelAnodeRearClamp.monitoring;
   "Unit1.EmNodes".emRelations.em06.cmControlNode.cmMendrelCathodeFrontClamp.monitoring := "Unit1.Em6.ControlNodes".cmMendrelCathodeFrontClamp.monitoring;
   "Unit1.EmNodes".emRelations.em06.cmControlNode.cmMendrelCathodeRearClamp.monitoring := "Unit1.Em6.ControlNodes".cmMendrelCathodeRearClamp.monitoring;
   "Unit1.EmNodes".emRelations.em06.cmControlNode.cmStackTableVaccum.monitoring := "Unit1.Em6.ControlNodes".cmStackTableVaccum.monitoring;
   "Unit1.EmNodes".emRelations.em06.cmControlNode.cmStackTableGapPadUpDown.monitoring := "Unit1.Em6.ControlNodes".cmStackTableGapPadUpDown.monitoring;
END_REGION

REGION Network 355: Em Relations Digital Signal
   RUNG wire#powerrail
      Move(in := "Unit1.Em6.ControlNodes".cmStackTableElectrodeDetect.monitoring, out1 => "Unit1.EmNodes".emRelations.em06.cmControlNode.cmStackTableElectrodeDetect.monitoring)
   END_RUNG
   // the same network as SCL:
   "Unit1.EmNodes".emRelations.em06.cmControlNode.cmStackTableElectrodeDetect.monitoring := "Unit1.Em6.ControlNodes".cmStackTableElectrodeDetect.monitoring;
END_REGION

REGION Network 356: Em Relations Select Job Status
   RUNG wire#powerrail
      Move(in := "Unit1.Em6.ControlNodes".stackTable.jobInterface.homeJob1, out1 => "Unit1.EmNodes".emRelations.em06.sequence.Spare1.jobInterface[1])
   END_RUNG
   // the same network as SCL:
   "Unit1.EmNodes".emRelations.em06.sequence.Spare1.jobInterface[1] := "Unit1.Em6.ControlNodes".stackTable.jobInterface.homeJob1;
END_REGION

REGION Network 357: Em Relations Sequence Interface
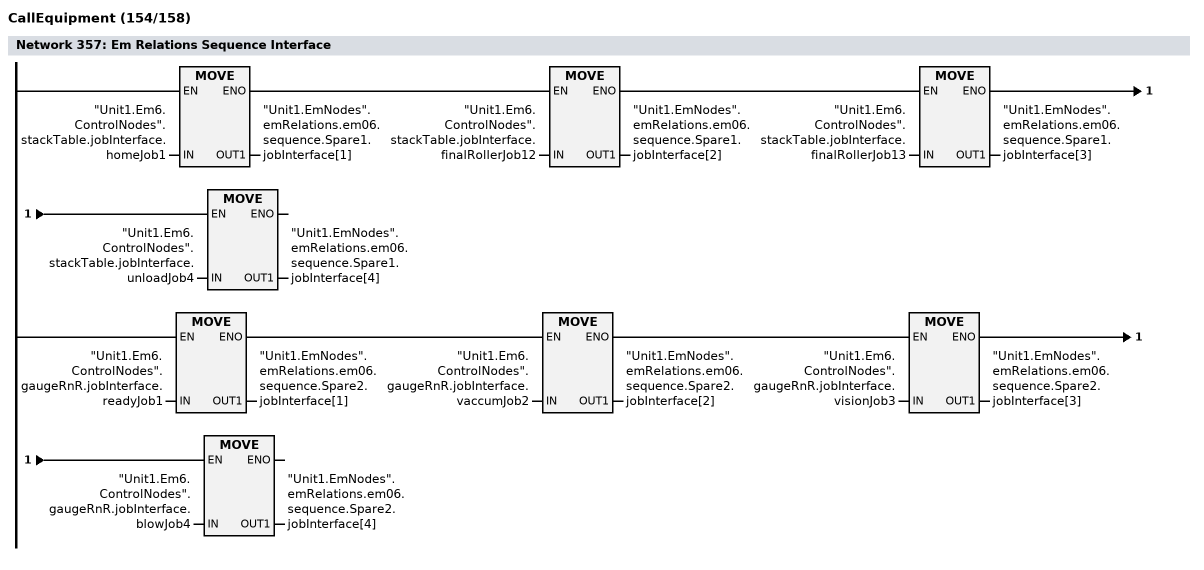
   RUNG wire#powerrail
      Move(in := "Unit1.Em6.ControlNodes".stackTable.jobInterface.homeJob1, out1 => "Unit1.EmNodes".emRelations.em06.sequence.Spare1.jobInterface[1])
      Move(in := "Unit1.Em6.ControlNodes".stackTable.jobInterface.finalRollerJob12, out1 => "Unit1.EmNodes".emRelations.em06.sequence.Spare1.jobInterface[2])
      Move(in := "Unit1.Em6.ControlNodes".stackTable.jobInterface.finalRollerJob13, out1 => "Unit1.EmNodes".emRelations.em06.sequence.Spare1.jobInterface[3])
      Move(in := "Unit1.Em6.ControlNodes".stackTable.jobInterface.unloadJob4, out1 => "Unit1.EmNodes".emRelations.em06.sequence.Spare1.jobInterface[4])
   END_RUNG
   RUNG wire#powerrail
      Move(in := "Unit1.Em6.ControlNodes".gaugeRnR.jobInterface.readyJob1, out1 => "Unit1.EmNodes".emRelations.em06.sequence.Spare2.jobInterface[1])
      Move(in := "Unit1.Em6.ControlNodes".gaugeRnR.jobInterface.vaccumJob2, out1 => "Unit1.EmNodes".emRelations.em06.sequence.Spare2.jobInterface[2])
      Move(in := "Unit1.Em6.ControlNodes".gaugeRnR.jobInterface.visionJob3, out1 => "Unit1.EmNodes".emRelations.em06.sequence.Spare2.jobInterface[3])
      Move(in := "Unit1.Em6.ControlNodes".gaugeRnR.jobInterface.blowJob4, out1 => "Unit1.EmNodes".emRelations.em06.sequence.Spare2.jobInterface[4])
   END_RUNG
   // the same network as SCL:
   "Unit1.EmNodes".emRelations.em06.sequence.Spare1.jobInterface[1] := "Unit1.Em6.ControlNodes".stackTable.jobInterface.homeJob1;
   "Unit1.EmNodes".emRelations.em06.sequence.Spare1.jobInterface[2] := "Unit1.Em6.ControlNodes".stackTable.jobInterface.finalRollerJob12;
   "Unit1.EmNodes".emRelations.em06.sequence.Spare1.jobInterface[3] := "Unit1.Em6.ControlNodes".stackTable.jobInterface.finalRollerJob13;
   "Unit1.EmNodes".emRelations.em06.sequence.Spare1.jobInterface[4] := "Unit1.Em6.ControlNodes".stackTable.jobInterface.unloadJob4;
   "Unit1.EmNodes".emRelations.em06.sequence.Spare2.jobInterface[1] := "Unit1.Em6.ControlNodes".gaugeRnR.jobInterface.readyJob1;
   "Unit1.EmNodes".emRelations.em06.sequence.Spare2.jobInterface[2] := "Unit1.Em6.ControlNodes".gaugeRnR.jobInterface.vaccumJob2;
   "Unit1.EmNodes".emRelations.em06.sequence.Spare2.jobInterface[3] := "Unit1.Em6.ControlNodes".gaugeRnR.jobInterface.visionJob3;
   "Unit1.EmNodes".emRelations.em06.sequence.Spare2.jobInterface[4] := "Unit1.Em6.ControlNodes".gaugeRnR.jobInterface.blowJob4;
END_REGION

REGION Network 358: Em Relations Softcam
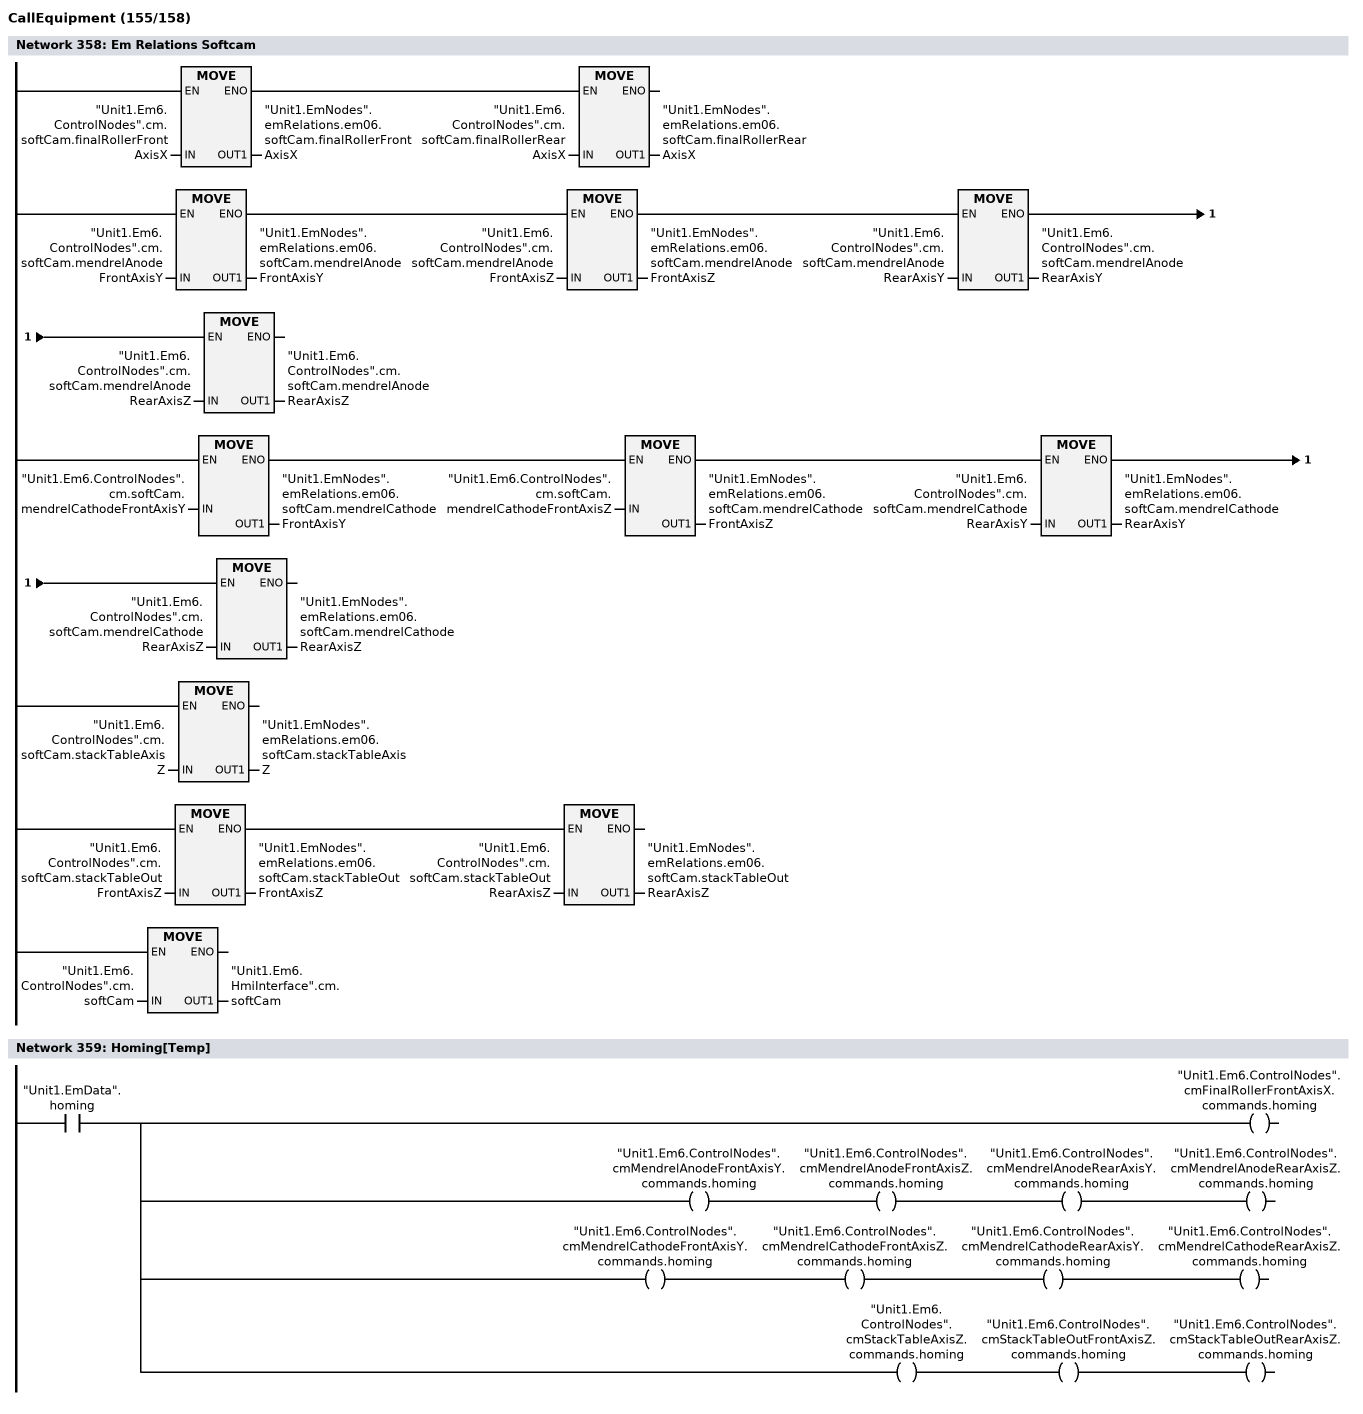
   RUNG wire#powerrail
      Move(in := "Unit1.Em6.ControlNodes".cm.softCam.finalRollerFrontAxisX, out1 => "Unit1.EmNodes".emRelations.em06.softCam.finalRollerFrontAxisX)
      Move(in := "Unit1.Em6.ControlNodes".cm.softCam.finalRollerRearAxisX, out1 => "Unit1.EmNodes".emRelations.em06.softCam.finalRollerRearAxisX)
   END_RUNG
   RUNG wire#powerrail
      Move(in := "Unit1.Em6.ControlNodes".cm.softCam.mendrelAnodeFrontAxisY, out1 => "Unit1.EmNodes".emRelations.em06.softCam.mendrelAnodeFrontAxisY)
      Move(in := "Unit1.Em6.ControlNodes".cm.softCam.mendrelAnodeFrontAxisZ, out1 => "Unit1.EmNodes".emRelations.em06.softCam.mendrelAnodeFrontAxisZ)
      Move(in := "Unit1.Em6.ControlNodes".cm.softCam.mendrelAnodeRearAxisY, out1 => "Unit1.Em6.ControlNodes".cm.softCam.mendrelAnodeRearAxisY)
      Move(in := "Unit1.Em6.ControlNodes".cm.softCam.mendrelAnodeRearAxisZ, out1 => "Unit1.Em6.ControlNodes".cm.softCam.mendrelAnodeRearAxisZ)
   END_RUNG
   RUNG wire#powerrail
      Move(in := "Unit1.Em6.ControlNodes".cm.softCam.mendrelCathodeFrontAxisY, out1 => "Unit1.EmNodes".emRelations.em06.softCam.mendrelCathodeFrontAxisY)
      Move(in := "Unit1.Em6.ControlNodes".cm.softCam.mendrelCathodeFrontAxisZ, out1 => "Unit1.EmNodes".emRelations.em06.softCam.mendrelCathodeFrontAxisZ)
      Move(in := "Unit1.Em6.ControlNodes".cm.softCam.mendrelCathodeRearAxisY, out1 => "Unit1.EmNodes".emRelations.em06.softCam.mendrelCathodeRearAxisY)
      Move(in := "Unit1.Em6.ControlNodes".cm.softCam.mendrelCathodeRearAxisZ, out1 => "Unit1.EmNodes".emRelations.em06.softCam.mendrelCathodeRearAxisZ)
   END_RUNG
   RUNG wire#powerrail
      Move(in := "Unit1.Em6.ControlNodes".cm.softCam.stackTableAxisZ, out1 => "Unit1.EmNodes".emRelations.em06.softCam.stackTableAxisZ)
   END_RUNG
   RUNG wire#powerrail
      Move(in := "Unit1.Em6.ControlNodes".cm.softCam.stackTableOutFrontAxisZ, out1 => "Unit1.EmNodes".emRelations.em06.softCam.stackTableOutFrontAxisZ)
      Move(in := "Unit1.Em6.ControlNodes".cm.softCam.stackTableOutRearAxisZ, out1 => "Unit1.EmNodes".emRelations.em06.softCam.stackTableOutRearAxisZ)
   END_RUNG
   RUNG wire#powerrail
      Move(in := "Unit1.Em6.ControlNodes".cm.softCam, out1 => "Unit1.Em6.HmiInterface".cm.softCam)
   END_RUNG
   // the same network as SCL:
   "Unit1.EmNodes".emRelations.em06.softCam.finalRollerFrontAxisX := "Unit1.Em6.ControlNodes".cm.softCam.finalRollerFrontAxisX;
   "Unit1.EmNodes".emRelations.em06.softCam.finalRollerRearAxisX := "Unit1.Em6.ControlNodes".cm.softCam.finalRollerRearAxisX;
   "Unit1.EmNodes".emRelations.em06.softCam.mendrelAnodeFrontAxisY := "Unit1.Em6.ControlNodes".cm.softCam.mendrelAnodeFrontAxisY;
   "Unit1.EmNodes".emRelations.em06.softCam.mendrelAnodeFrontAxisZ := "Unit1.Em6.ControlNodes".cm.softCam.mendrelAnodeFrontAxisZ;
   "Unit1.Em6.ControlNodes".cm.softCam.mendrelAnodeRearAxisY := "Unit1.Em6.ControlNodes".cm.softCam.mendrelAnodeRearAxisY;
   "Unit1.Em6.ControlNodes".cm.softCam.mendrelAnodeRearAxisZ := "Unit1.Em6.ControlNodes".cm.softCam.mendrelAnodeRearAxisZ;
   "Unit1.EmNodes".emRelations.em06.softCam.mendrelCathodeFrontAxisY := "Unit1.Em6.ControlNodes".cm.softCam.mendrelCathodeFrontAxisY;
   "Unit1.EmNodes".emRelations.em06.softCam.mendrelCathodeFrontAxisZ := "Unit1.Em6.ControlNodes".cm.softCam.mendrelCathodeFrontAxisZ;
   "Unit1.EmNodes".emRelations.em06.softCam.mendrelCathodeRearAxisY := "Unit1.Em6.ControlNodes".cm.softCam.mendrelCathodeRearAxisY;
   "Unit1.EmNodes".emRelations.em06.softCam.mendrelCathodeRearAxisZ := "Unit1.Em6.ControlNodes".cm.softCam.mendrelCathodeRearAxisZ;
   "Unit1.EmNodes".emRelations.em06.softCam.stackTableAxisZ := "Unit1.Em6.ControlNodes".cm.softCam.stackTableAxisZ;
   "Unit1.EmNodes".emRelations.em06.softCam.stackTableOutFrontAxisZ := "Unit1.Em6.ControlNodes".cm.softCam.stackTableOutFrontAxisZ;
   "Unit1.EmNodes".emRelations.em06.softCam.stackTableOutRearAxisZ := "Unit1.Em6.ControlNodes".cm.softCam.stackTableOutRearAxisZ;
   "Unit1.Em6.HmiInterface".cm.softCam := "Unit1.Em6.ControlNodes".cm.softCam;
END_REGION

REGION Network 359: Homing[Temp]
   RUNG wire#powerrail
      Contact( "Unit1.EmData".homing )
      wire#w1
      Coil( "Unit1.Em6.ControlNodes".cmFinalRollerFrontAxisX.commands.homing )
   END_RUNG
   RUNG wire#w1
      Coil( "Unit1.Em6.ControlNodes".cmMendrelAnodeFrontAxisY.commands.homing )
      Coil( "Unit1.Em6.ControlNodes".cmMendrelAnodeFrontAxisZ.commands.homing )
      Coil( "Unit1.Em6.ControlNodes".cmMendrelAnodeRearAxisY.commands.homing )
      Coil( "Unit1.Em6.ControlNodes".cmMendrelAnodeRearAxisZ.commands.homing )
   END_RUNG
   RUNG wire#w1
      Coil( "Unit1.Em6.ControlNodes".cmMendrelCathodeFrontAxisY.commands.homing )
      Coil( "Unit1.Em6.ControlNodes".cmMendrelCathodeFrontAxisZ.commands.homing )
      Coil( "Unit1.Em6.ControlNodes".cmMendrelCathodeRearAxisY.commands.homing )
      Coil( "Unit1.Em6.ControlNodes".cmMendrelCathodeRearAxisZ.commands.homing )
   END_RUNG
   RUNG wire#w1
      Coil( "Unit1.Em6.ControlNodes".cmStackTableAxisZ.commands.homing )
      Coil( "Unit1.Em6.ControlNodes".cmStackTableOutFrontAxisZ.commands.homing )
      Coil( "Unit1.Em6.ControlNodes".cmStackTableOutRearAxisZ.commands.homing )
   END_RUNG
   // the same network as SCL:
   "Unit1.Em6.ControlNodes".cmFinalRollerFrontAxisX.commands.homing := "Unit1.EmData".homing;
   "Unit1.Em6.ControlNodes".cmMendrelAnodeFrontAxisY.commands.homing := "Unit1.EmData".homing;
   "Unit1.Em6.ControlNodes".cmMendrelAnodeFrontAxisZ.commands.homing := "Unit1.EmData".homing;
   "Unit1.Em6.ControlNodes".cmMendrelAnodeRearAxisY.commands.homing := "Unit1.EmData".homing;
   "Unit1.Em6.ControlNodes".cmMendrelAnodeRearAxisZ.commands.homing := "Unit1.EmData".homing;
   "Unit1.Em6.ControlNodes".cmMendrelCathodeFrontAxisY.commands.homing := "Unit1.EmData".homing;
   "Unit1.Em6.ControlNodes".cmMendrelCathodeFrontAxisZ.commands.homing := "Unit1.EmData".homing;
   "Unit1.Em6.ControlNodes".cmMendrelCathodeRearAxisY.commands.homing := "Unit1.EmData".homing;
   "Unit1.Em6.ControlNodes".cmMendrelCathodeRearAxisZ.commands.homing := "Unit1.EmData".homing;
   "Unit1.Em6.ControlNodes".cmStackTableAxisZ.commands.homing := "Unit1.EmData".homing;
   "Unit1.Em6.ControlNodes".cmStackTableOutFrontAxisZ.commands.homing := "Unit1.EmData".homing;
   "Unit1.Em6.ControlNodes".cmStackTableOutRearAxisZ.commands.homing := "Unit1.EmData".homing;
END_REGION

REGION Network 360: Stack PartStatus Data handle
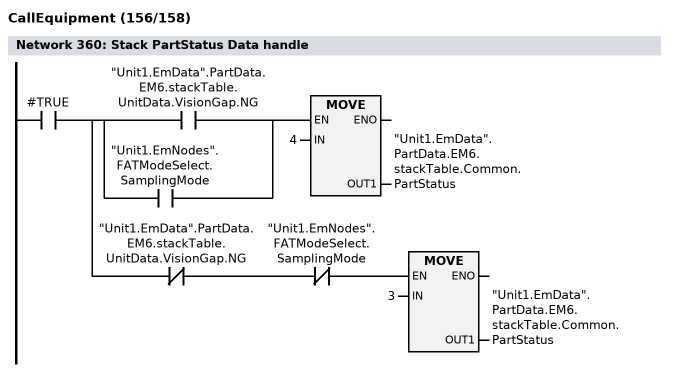
   RUNG wire#powerrail
      Contact( #TRUE )
      wire#w1
      Contact( "Unit1.EmData".PartData.EM6.stackTable.UnitData.VisionGap.NG )
      wire#w2
      Move(in := 4, out1 => "Unit1.EmData".PartData.EM6.stackTable.Common.PartStatus)
   END_RUNG
   RUNG wire#w1
      Contact( "Unit1.EmNodes".FATModeSelect.SamplingMode )
   END_RUNG wire#w2
   RUNG wire#w1
      I_Contact( "Unit1.EmData".PartData.EM6.stackTable.UnitData.VisionGap.NG )
      I_Contact( "Unit1.EmNodes".FATModeSelect.SamplingMode )
      Move(in := 3, out1 => "Unit1.EmData".PartData.EM6.stackTable.Common.PartStatus)
   END_RUNG
   // the same network as SCL:
   IF #TRUE AND ("Unit1.EmData".PartData.EM6.stackTable.UnitData.VisionGap.NG OR "Unit1.EmNodes".FATModeSelect.SamplingMode) THEN
       "Unit1.EmData".PartData.EM6.stackTable.Common.PartStatus := 4;
   END_IF;
   IF #TRUE AND NOT "Unit1.EmData".PartData.EM6.stackTable.UnitData.VisionGap.NG AND NOT "Unit1.EmNodes".FATModeSelect.SamplingMode THEN
       "Unit1.EmData".PartData.EM6.stackTable.Common.PartStatus := 3;
   END_IF;
END_REGION

REGION Network 362 (SCL): SyncMotion Configuration
   "Unit1.MotionNodes".PLCToMotion.TechnologyObject.Axis.FinalRoller := "BA040AZSCDR21_FinalRollerFrontAxisX";
   "Unit1.MotionNodes".PLCToMotion.TechnologyObject.Axis.AnodeMandrelYFront := "BA040AZSCDR23_MendrelAnodeFrontAxisY";
   "Unit1.MotionNodes".PLCToMotion.TechnologyObject.Axis.AnodeMandrelYRear := "BA040AZSCDR25_MendrelAnodeRearAxisY";
   "Unit1.MotionNodes".PLCToMotion.TechnologyObject.Axis.AnodeMandrelZFront := "BA040AZSCDR24_MendrelAnodeFrontAxisZ";
   "Unit1.MotionNodes".PLCToMotion.TechnologyObject.Axis.AnodeMandrelZRear := "BA040AZSCDR26_MendrelAnodeRearAxisZ";
   "Unit1.MotionNodes".PLCToMotion.TechnologyObject.Axis.CathodeMandrelYFront := "BA040AZSCDR27_MendrelCathodeFrontAxisY";
   "Unit1.MotionNodes".PLCToMotion.TechnologyObject.Axis.CathodeMandrelYRear := "BA040AZSCDR29_MendrelCathodeRearAxisY";
   "Unit1.MotionNodes".PLCToMotion.TechnologyObject.Axis.CathodeMandrelZFront := "BA040AZSCDR28_MendrelCathodeFrontAxisZ";
   "Unit1.MotionNodes".PLCToMotion.TechnologyObject.Axis.CathodeMandrelZRear := "BA040AZSCDR30_MendrelCathodeRearAxisZ";
   "Unit1.MotionNodes".PLCToMotion.TechnologyObject.Axis.MasterVirtual := "BA040A_MasterAxis";


   "Unit1.Em6.Config".outputCam[1] := "FinalRollerXFwd";
   "Unit1.Em6.Config".outputCam[2] := "FinalRollerXBwd";
   "Unit1.Em6.Config".outputCam[3] := "FinalRollerXStackTableDown";
   "Unit1.Em6.Config".outputCam[4] := "FinalRollerXStackAnodeVision";
   "Unit1.Em6.Config".outputCam[5] := "FinalRollerXStackCathodeVision";


   "Unit1.MotionNodes".PLCToMotion.TechnologyObject.OutputCam.FinalRollerXFwdOutputCam := "Unit1.Em6.Config".outputCam[1];
   "Unit1.MotionNodes".PLCToMotion.TechnologyObject.OutputCam.FinalRollerXBwdOutputCam := "Unit1.Em6.Config".outputCam[2];
   "Unit1.MotionNodes".PLCToMotion.TechnologyObject.OutputCam.FinalRollerXStackTableDownOutputCam := "Unit1.Em6.Config".outputCam[3];
   "Unit1.MotionNodes".PLCToMotion.TechnologyObject.OutputCam.FinalRollerXStackAnodeVisionOutputCam := "Unit1.Em6.Config".outputCam[4];
   "Unit1.MotionNodes".PLCToMotion.TechnologyObject.OutputCam.FinalRollerXStackCathodeVisionOutputCam := "Unit1.Em6.Config".outputCam[5];


   // _.Unit1.SyncMotion.Configuration.TechnologyObjects.StackMain.Cam.FinalRollerCam := Config.cam[1];
   // _.Unit1.SyncMotion.Configuration.TechnologyObjects.StackMain.Cam.AnodeMandrelYFrontCam := Config.cam[2];
   // _.Unit1.SyncMotion.Configuration.TechnologyObjects.StackMain.Cam.AnodeMandrelYRearCam := Config.cam[3];
   // _.Unit1.SyncMotion.Configuration.TechnologyObjects.StackMain.Cam.AnodeMandrelZFrontCam := Config.cam[4];
   // _.Unit1.SyncMotion.Configuration.TechnologyObjects.StackMain.Cam.AnodeMandrelZRearCam := Config.cam[5];
   // _.Unit1.SyncMotion.Configuration.TechnologyObjects.StackMain.Cam.CathodeMandrelYFrontCam := Config.cam[6];
   // _.Unit1.SyncMotion.Configuration.TechnologyObjects.StackMain.Cam.CathodeMandrelYRearCam := Config.cam[7];
   // _.Unit1.SyncMotion.Configuration.TechnologyObjects.StackMain.Cam.CathodeMandrelZFrontCam := Config.cam[8];
   // _.Unit1.SyncMotion.Configuration.TechnologyObjects.StackMain.Cam.CathodeMandrelZRearCam := Config.cam[9];
END_REGION

REGION Network 363: Axis
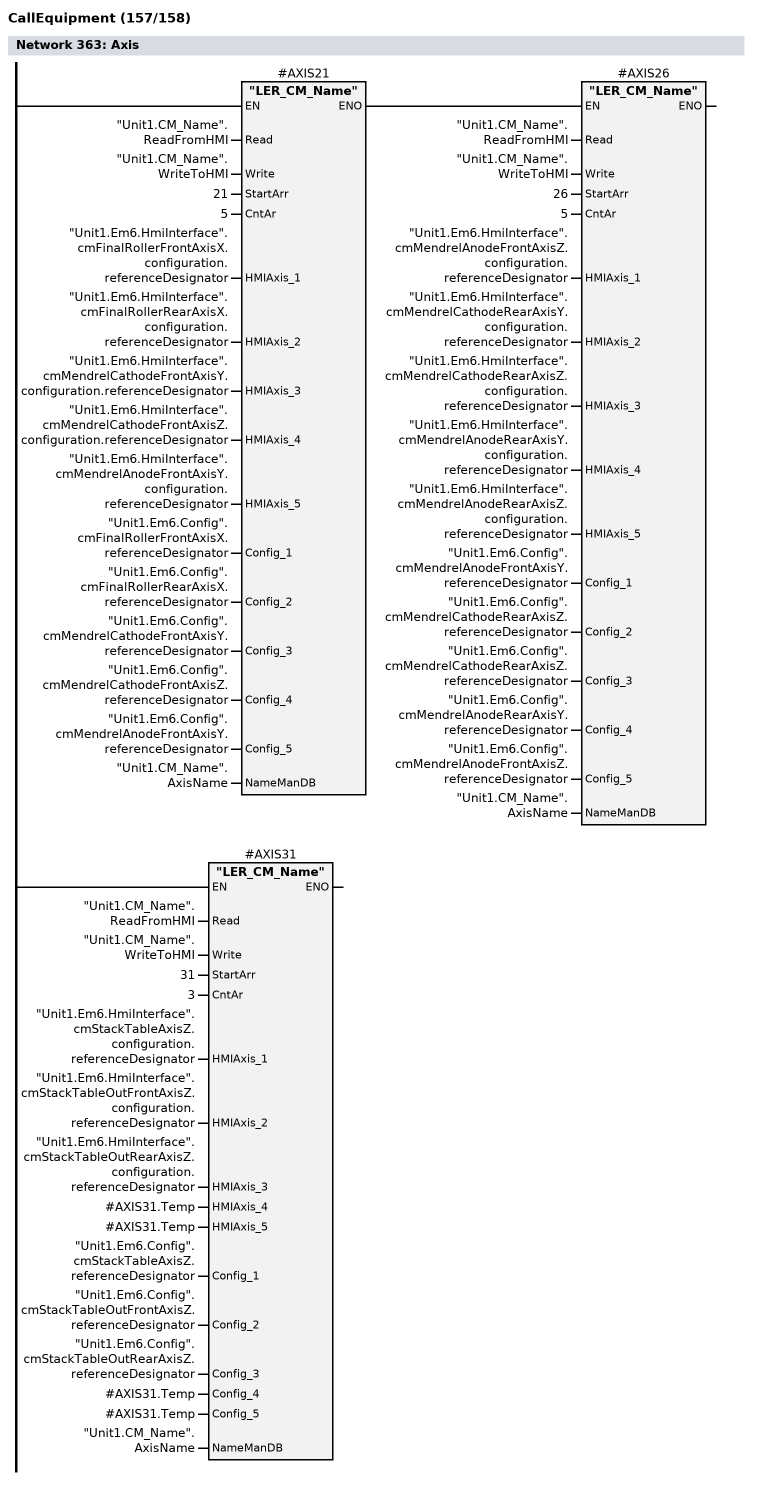
   RUNG wire#powerrail
      #AXIS21(Read := "Unit1.CM_Name".ReadFromHMI, Write := "Unit1.CM_Name".WriteToHMI, StartArr := 21, CntAr := 5, HMIAxis_1 := "Unit1.Em6.HmiInterface".cmFinalRollerFrontAxisX.configuration.referenceDesignator, HMIAxis_2 := "Unit1.Em6.HmiInterface".cmFinalRollerRearAxisX.configuration.referenceDesignator, HMIAxis_3 := "Unit1.Em6.HmiInterface".cmMendrelCathodeFrontAxisY.configuration.referenceDesignator, HMIAxis_4 := "Unit1.Em6.HmiInterface".cmMendrelCathodeFrontAxisZ.configuration.referenceDesignator, HMIAxis_5 := "Unit1.Em6.HmiInterface".cmMendrelAnodeFrontAxisY.configuration.referenceDesignator, Config_1 := "Unit1.Em6.Config".cmFinalRollerFrontAxisX.referenceDesignator, Config_2 := "Unit1.Em6.Config".cmFinalRollerRearAxisX.referenceDesignator, Config_3 := "Unit1.Em6.Config".cmMendrelCathodeFrontAxisY.referenceDesignator, Config_4 := "Unit1.Em6.Config".cmMendrelCathodeFrontAxisZ.referenceDesignator, Config_5 := "Unit1.Em6.Config".cmMendrelAnodeFrontAxisY.referenceDesignator, NameManDB := "Unit1.CM_Name".AxisName)
      #AXIS26(Read := "Unit1.CM_Name".ReadFromHMI, Write := "Unit1.CM_Name".WriteToHMI, StartArr := 26, CntAr := 5, HMIAxis_1 := "Unit1.Em6.HmiInterface".cmMendrelAnodeFrontAxisZ.configuration.referenceDesignator, HMIAxis_2 := "Unit1.Em6.HmiInterface".cmMendrelCathodeRearAxisY.configuration.referenceDesignator, HMIAxis_3 := "Unit1.Em6.HmiInterface".cmMendrelCathodeRearAxisZ.configuration.referenceDesignator, HMIAxis_4 := "Unit1.Em6.HmiInterface".cmMendrelAnodeRearAxisY.configuration.referenceDesignator, HMIAxis_5 := "Unit1.Em6.HmiInterface".cmMendrelAnodeRearAxisZ.configuration.referenceDesignator, Config_1 := "Unit1.Em6.Config".cmMendrelAnodeFrontAxisY.referenceDesignator, Config_2 := "Unit1.Em6.Config".cmMendrelCathodeRearAxisZ.referenceDesignator, Config_3 := "Unit1.Em6.Config".cmMendrelCathodeRearAxisZ.referenceDesignator, Config_4 := "Unit1.Em6.Config".cmMendrelAnodeRearAxisY.referenceDesignator, Config_5 := "Unit1.Em6.Config".cmMendrelAnodeFrontAxisZ.referenceDesignator, NameManDB := "Unit1.CM_Name".AxisName)
   END_RUNG
   RUNG wire#powerrail
      #AXIS31(Read := "Unit1.CM_Name".ReadFromHMI, Write := "Unit1.CM_Name".WriteToHMI, StartArr := 31, CntAr := 3, HMIAxis_1 := "Unit1.Em6.HmiInterface".cmStackTableAxisZ.configuration.referenceDesignator, HMIAxis_2 := "Unit1.Em6.HmiInterface".cmStackTableOutFrontAxisZ.configuration.referenceDesignator, HMIAxis_3 := "Unit1.Em6.HmiInterface".cmStackTableOutRearAxisZ.configuration.referenceDesignator, HMIAxis_4 := #AXIS31.Temp, HMIAxis_5 := #AXIS31.Temp, Config_1 := "Unit1.Em6.Config".cmStackTableAxisZ.referenceDesignator, Config_2 := "Unit1.Em6.Config".cmStackTableOutFrontAxisZ.referenceDesignator, Config_3 := "Unit1.Em6.Config".cmStackTableOutRearAxisZ.referenceDesignator, Config_4 := #AXIS31.Temp, Config_5 := #AXIS31.Temp, NameManDB := "Unit1.CM_Name".AxisName)
   END_RUNG
   // the same network as SCL:
   #AXIS21(Read := "Unit1.CM_Name".ReadFromHMI,   // "LER_CM_Name"
           Write := "Unit1.CM_Name".WriteToHMI,
           StartArr := 21,
           CntAr := 5,
           HMIAxis_1 := "Unit1.Em6.HmiInterface".cmFinalRollerFrontAxisX.configuration.referenceDesignator,
           HMIAxis_2 := "Unit1.Em6.HmiInterface".cmFinalRollerRearAxisX.configuration.referenceDesignator,
           HMIAxis_3 := "Unit1.Em6.HmiInterface".cmMendrelCathodeFrontAxisY.configuration.referenceDesignator,
           HMIAxis_4 := "Unit1.Em6.HmiInterface".cmMendrelCathodeFrontAxisZ.configuration.referenceDesignator,
           HMIAxis_5 := "Unit1.Em6.HmiInterface".cmMendrelAnodeFrontAxisY.configuration.referenceDesignator,
           Config_1 := "Unit1.Em6.Config".cmFinalRollerFrontAxisX.referenceDesignator,
           Config_2 := "Unit1.Em6.Config".cmFinalRollerRearAxisX.referenceDesignator,
           Config_3 := "Unit1.Em6.Config".cmMendrelCathodeFrontAxisY.referenceDesignator,
           Config_4 := "Unit1.Em6.Config".cmMendrelCathodeFrontAxisZ.referenceDesignator,
           Config_5 := "Unit1.Em6.Config".cmMendrelAnodeFrontAxisY.referenceDesignator,
           NameManDB := "Unit1.CM_Name".AxisName,
           ENO => #_w1);
   IF #_w1 THEN
       #AXIS26(Read := "Unit1.CM_Name".ReadFromHMI,   // "LER_CM_Name"
               Write := "Unit1.CM_Name".WriteToHMI,
               StartArr := 26,
               CntAr := 5,
               HMIAxis_1 := "Unit1.Em6.HmiInterface".cmMendrelAnodeFrontAxisZ.configuration.referenceDesignator,
               HMIAxis_2 := "Unit1.Em6.HmiInterface".cmMendrelCathodeRearAxisY.configuration.referenceDesignator,
               HMIAxis_3 := "Unit1.Em6.HmiInterface".cmMendrelCathodeRearAxisZ.configuration.referenceDesignator,
               HMIAxis_4 := "Unit1.Em6.HmiInterface".cmMendrelAnodeRearAxisY.configuration.referenceDesignator,
               HMIAxis_5 := "Unit1.Em6.HmiInterface".cmMendrelAnodeRearAxisZ.configuration.referenceDesignator,
               Config_1 := "Unit1.Em6.Config".cmMendrelAnodeFrontAxisY.referenceDesignator,
               Config_2 := "Unit1.Em6.Config".cmMendrelCathodeRearAxisZ.referenceDesignator,
               Config_3 := "Unit1.Em6.Config".cmMendrelCathodeRearAxisZ.referenceDesignator,
               Config_4 := "Unit1.Em6.Config".cmMendrelAnodeRearAxisY.referenceDesignator,
               Config_5 := "Unit1.Em6.Config".cmMendrelAnodeFrontAxisZ.referenceDesignator,
               NameManDB := "Unit1.CM_Name".AxisName);
   END_IF;
   #AXIS31(Read := "Unit1.CM_Name".ReadFromHMI,   // "LER_CM_Name"
           Write := "Unit1.CM_Name".WriteToHMI,
           StartArr := 31,
           CntAr := 3,
           HMIAxis_1 := "Unit1.Em6.HmiInterface".cmStackTableAxisZ.configuration.referenceDesignator,
           HMIAxis_2 := "Unit1.Em6.HmiInterface".cmStackTableOutFrontAxisZ.configuration.referenceDesignator,
           HMIAxis_3 := "Unit1.Em6.HmiInterface".cmStackTableOutRearAxisZ.configuration.referenceDesignator,
           HMIAxis_4 := #AXIS31.Temp,
           HMIAxis_5 := #AXIS31.Temp,
           Config_1 := "Unit1.Em6.Config".cmStackTableAxisZ.referenceDesignator,
           Config_2 := "Unit1.Em6.Config".cmStackTableOutFrontAxisZ.referenceDesignator,
           Config_3 := "Unit1.Em6.Config".cmStackTableOutRearAxisZ.referenceDesignator,
           Config_4 := #AXIS31.Temp,
           Config_5 := #AXIS31.Temp,
           NameManDB := "Unit1.CM_Name".AxisName);
END_REGION

REGION Network 364: Cylinder
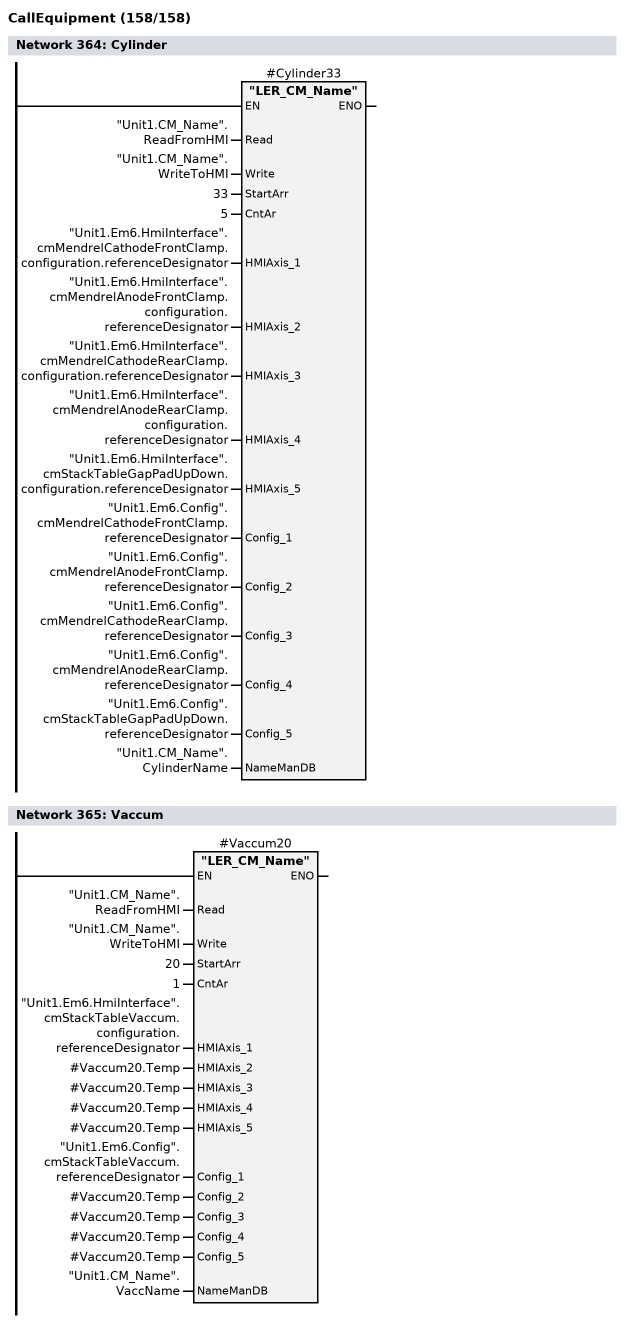
   RUNG wire#powerrail
      #Cylinder33(Read := "Unit1.CM_Name".ReadFromHMI, Write := "Unit1.CM_Name".WriteToHMI, StartArr := 33, CntAr := 5, HMIAxis_1 := "Unit1.Em6.HmiInterface".cmMendrelCathodeFrontClamp.configuration.referenceDesignator, HMIAxis_2 := "Unit1.Em6.HmiInterface".cmMendrelAnodeFrontClamp.configuration.referenceDesignator, HMIAxis_3 := "Unit1.Em6.HmiInterface".cmMendrelCathodeRearClamp.configuration.referenceDesignator, HMIAxis_4 := "Unit1.Em6.HmiInterface".cmMendrelAnodeRearClamp.configuration.referenceDesignator, HMIAxis_5 := "Unit1.Em6.HmiInterface".cmStackTableGapPadUpDown.configuration.referenceDesignator, Config_1 := "Unit1.Em6.Config".cmMendrelCathodeFrontClamp.referenceDesignator, Config_2 := "Unit1.Em6.Config".cmMendrelAnodeFrontClamp.referenceDesignator, Config_3 := "Unit1.Em6.Config".cmMendrelCathodeRearClamp.referenceDesignator, Config_4 := "Unit1.Em6.Config".cmMendrelAnodeRearClamp.referenceDesignator, Config_5 := "Unit1.Em6.Config".cmStackTableGapPadUpDown.referenceDesignator, NameManDB := "Unit1.CM_Name".CylinderName)
   END_RUNG
   // the same network as SCL:
   #Cylinder33(Read := "Unit1.CM_Name".ReadFromHMI,   // "LER_CM_Name"
               Write := "Unit1.CM_Name".WriteToHMI,
               StartArr := 33,
               CntAr := 5,
               HMIAxis_1 := "Unit1.Em6.HmiInterface".cmMendrelCathodeFrontClamp.configuration.referenceDesignator,
               HMIAxis_2 := "Unit1.Em6.HmiInterface".cmMendrelAnodeFrontClamp.configuration.referenceDesignator,
               HMIAxis_3 := "Unit1.Em6.HmiInterface".cmMendrelCathodeRearClamp.configuration.referenceDesignator,
               HMIAxis_4 := "Unit1.Em6.HmiInterface".cmMendrelAnodeRearClamp.configuration.referenceDesignator,
               HMIAxis_5 := "Unit1.Em6.HmiInterface".cmStackTableGapPadUpDown.configuration.referenceDesignator,
               Config_1 := "Unit1.Em6.Config".cmMendrelCathodeFrontClamp.referenceDesignator,
               Config_2 := "Unit1.Em6.Config".cmMendrelAnodeFrontClamp.referenceDesignator,
               Config_3 := "Unit1.Em6.Config".cmMendrelCathodeRearClamp.referenceDesignator,
               Config_4 := "Unit1.Em6.Config".cmMendrelAnodeRearClamp.referenceDesignator,
               Config_5 := "Unit1.Em6.Config".cmStackTableGapPadUpDown.referenceDesignator,
               NameManDB := "Unit1.CM_Name".CylinderName);
END_REGION

REGION Network 365: Vaccum
   RUNG wire#powerrail
      #Vaccum20(Read := "Unit1.CM_Name".ReadFromHMI, Write := "Unit1.CM_Name".WriteToHMI, StartArr := 20, CntAr := 1, HMIAxis_1 := "Unit1.Em6.HmiInterface".cmStackTableVaccum.configuration.referenceDesignator, HMIAxis_2 := #Vaccum20.Temp, HMIAxis_3 := #Vaccum20.Temp, HMIAxis_4 := #Vaccum20.Temp, HMIAxis_5 := #Vaccum20.Temp, Config_1 := "Unit1.Em6.Config".cmStackTableVaccum.referenceDesignator, Config_2 := #Vaccum20.Temp, Config_3 := #Vaccum20.Temp, Config_4 := #Vaccum20.Temp, Config_5 := #Vaccum20.Temp, NameManDB := "Unit1.CM_Name".VaccName)
   END_RUNG
   // the same network as SCL:
   #Vaccum20(Read := "Unit1.CM_Name".ReadFromHMI,   // "LER_CM_Name"
             Write := "Unit1.CM_Name".WriteToHMI,
             StartArr := 20,
             CntAr := 1,
             HMIAxis_1 := "Unit1.Em6.HmiInterface".cmStackTableVaccum.configuration.referenceDesignator,
             HMIAxis_2 := #Vaccum20.Temp,
             HMIAxis_3 := #Vaccum20.Temp,
             HMIAxis_4 := #Vaccum20.Temp,
             HMIAxis_5 := #Vaccum20.Temp,
             Config_1 := "Unit1.Em6.Config".cmStackTableVaccum.referenceDesignator,
             Config_2 := #Vaccum20.Temp,
             Config_3 := #Vaccum20.Temp,
             Config_4 := #Vaccum20.Temp,
             Config_5 := #Vaccum20.Temp,
             NameManDB := "Unit1.CM_Name".VaccName);
END_REGION
END_FUNCTION_BLOCK
